// TwinCAT 3 PLC project UtilitiesLib
// Title: IBF_Utilities
// Company: Industrial Brains B.V.
// ProjectVersion: 2.0.0.0
// Description: Utilities library contains all basic utilities needed like system variables, messages, parameters etc.
// ProgramVersion: 3.1.4022.4
// libraries:
//   Tc2_Standard, * (Beckhoff Automation GmbH)
//   Tc2_System, * (Beckhoff Automation GmbH)
//   Tc2_Utilities, * (Beckhoff Automation GmbH)
//   Tc3_EventLogger, * (Beckhoff Automation GmbH)
//   Tc3_Module, * (Beckhoff Automation GmbH)
// project tree:
//   Avarage/ FB_RollingAverageLREAL.TcPOU, FB_RollingAverageTime.TcPOU, F_AverageLREAL.TcPOU, F_AverageTime.TcPOU
//   BaseFunctions/ FB_Base.TcPOU, FB_Base_WithEvent.TcPOU, FB_FunctionBase.TcPOU, FB_FunctionBase_WIthEvent.TcPOU
//   Compare/Functions/ Between.TcPOU, Between360deg.TcPOU
//   Conversion/ DegS_To_Rpm.TcPOU, DegS_To_Rpm_And_MMin.TcPOU, Grey_To_Bin.TcPOU, MMin_To_Rpm_And_DegS.TcPOU, Rpm_To_DegS.TcPOU
//   FaultsAndMessages/Functions/ FB_EventHandler.TcPOU, Fb_FaultHandler.TcPOU, FB_OperatorMessageDisplay.TcPOU
//   General/DataTypes/ Udt_TimerBandwith.TcDUT
//   GVLs/ DataManager.TcGVL, GVL_FixedValues.TcGVL, GVL_Message.TcGVL, GVL_Parameters.TcGVL, Sys_Variables.TcGVL
//   FaultsAndMessages/DataTypes/ E_ComponentTypes.TcTLEO, E_Locations.TcTLEO, E_MessageNumbers.TcTLEO, E_FaultTypes.TcTLEO, UDT_Fault.TcDUT
//   FaultsAndMessages/ Param_Messages.TcGVL
//   MovePathCalculations/ fAccDecCalc.TcPOU (not stored)
//   Parameter/DataTypes/Old/ UDT_Parameter_1.TcDUT, Udt_ParameterRetain.TcDUT, Udt_Parameter_2.TcDUT, Udt_ParLog_Old.TcDUT
//   Parameter/DataTypes/ Udt_ParameterId.TcDUT, Udt_Parameter.TcDUT
//   Parameter/Functions/ FB_ParameterHandler.TcPOU, Fb_ParLogging.TcPOU, F_ParToCsvLine.TcPOU
//   PathFunctions/ F_FBNameFromPath.TcPOU, F_GetLevelFromPath.TcPOU
//   Positions/FunctionBlocks/ FB_PositionTrigger_Old.TcPOU, FB_PositionTrigger.TcPOU
//   Positions/Functions/ F_AccDecDistanceFromTime.TcPOU, F_AccDecDistanceFromVelo.TcPOU, F_PosCheck.TcPOU, F_TopVelocityFromTime.TcPOU, F_TriggerPosOffset.TcPOU
//   StepFunctions/ FB_CycleTrigger.TcPOU (not stored), FB_Step.TcPOU
//   System/Functions/DataManagement/ FB_PersistentDataManager.TcPOU
//   System/Functions/ Fb_SystemVariables.TcPOU
//   / Utilities_CD.TcCD (not stored)

// ---- General/DataTypes/Udt_TimerBandwith.TcDUT
TYPE Udt_TimerBandwith :
STRUCT
	Minimal	:LREAL;// Timer values, Minimum time
	Nominal	:LREAL;// timer values, nominal time
	Maximum	:LREAL;// Timer values, Maximum time
END_STRUCT
END_TYPE

// ---- FaultsAndMessages/DataTypes/E_ComponentTypes.TcTLEO
{attribute 'qualified_only'}
{attribute 'strict'}
{attribute 'to_string'}
TYPE E_ComponentTypes :
(
	// No entry
		NA			:= 0,
	// Actuators 
		Cylinder 	:= 10,
		Axis		:= 11,
		Heaters		:= 12,
	// Buttons 
		EstopButton	:= 20,
		EstopBumper	:= 21,	
		Pushbutton 	:= 22,
		Switch		:= 23,
	// I/O
		SafeIO		:= 30,
		Rio_Box		:= 31,
		Rio_Slot	:= 32,
		Encoder		:= 33,
		DiInput		:= 34,
		AnInput		:= 35,
		DiOutput	:= 36,
		AnOutput	:= 37,
	// Drive
		ServoDrive 	:= 40,
	// Operation
		HMI			:= 50,
		RemoteOS	:= 51,
		RemoteDB	:= 52,
	// Assemblies
		Assembly 	:= 60,
		SubAssembly	:= 61,
	// functions
		MainProgram		:= 100,
		StepProgram		:= 101,
		FunctionBlock	:= 102 
)UDINT;
END_TYPE

// ---- FaultsAndMessages/DataTypes/E_Locations.TcTLEO
{attribute 'qualified_only'}
{attribute 'strict'}
TYPE E_Locations :
(
	MainPLC,
	MainPower_230V, 
	MainPower_24V, 
	MainAirSupply,
	MainScreen,
	MainIO,
	RemoteIO
);
END_TYPE

// ---- FaultsAndMessages/DataTypes/E_MessageNumbers.TcTLEO
{attribute 'qualified_only'}
{attribute 'strict'}
TYPE E_MessageNumbers :
(
	// no messages
		NA_NoMessage		:= 0, // no message active
	// System faults
		FF_Unknown 			:= 1, // unknown error occured 
		FF_NoCommunication 	:= 2, // no communication detected
		FF_ComunicationFault:= 3, // Communication error detected (does not match expected com)
		FF_Overload			:= 4, // hardware overload detected
		FF_EncoderFault		:= 5, // encoder signal incorrect or not present
		FF_SlaveFault		:= 6, // slave system is has active fatal fault
		FF_AxisFault		:= 7, // Axis fault feedback
		FF_DriveFault		:= 8, // Axis drive fault
		FF_Collision		:= 9, // Collision detected between 2 or more parts of the machine
	// Hardware faults
		CF_FeedbackFault		:= 100,	// Hardware feedback is does not match expected
		CF_WrongDirection		:= 101, // Hardware moving in incorrect direction
		CF_MoveToFast			:= 102, // Hardware movement completion time is lower then minimum
		CF_MoveToSlow			:= 103, // hardware movement maximum time was exceeded
		CF_WrongPosition		:= 104,	// Hardware is at different position then expected
		CF_Obstruction			:= 105, // Obstruction detected in movement path
	// Missing conditions
		MC_WaitingForproduct	:= 200,	// Waiting for product
		MC_WaitingForOperator	:= 201, // Waiting for operator action
		MC_WaitingForModule		:= 202,	// Waiting for other module
		MC_WaitingForMaster		:= 203, // Waiting Waiting for master
		MC_WaitingForSlave		:= 204, // waiting for slave
		MC_WrongPosition		:= 205, // Action or command not possible in current position
	// Operator messages
		OM_AlmostEmpty			:= 300, // product is almost empty refil is required
		OM_Finished 			:= 301, // product or action is finished
		OM_ready				:= 302, // ready for new task
	// Test Messages
		FF_MessageTest			:= 900, // Fatal fault message test
		CF_MessageTest			:= 901, // Cycle fault message test
		MC_MessageTest			:= 902, // Missing condition message test
		OM_MessageTest			:= 903	// Operator message test
)UDINT;
END_TYPE

// ---- FaultsAndMessages/DataTypes/E_FaultTypes.TcTLEO
{attribute 'qualified_only'}
{attribute 'strict'}
{attribute 'to_string'}
TYPE E_FaultTypes :
(
	NA	:= 0, // Not applicable
	OM 	:= 1, // Operator message
	MC	:= 2, // Missing condition
	CF	:= 3, // Cycle Fault
	FF	:= 4, // Fatal fault
	OW  := 5  // Operator warning
)UDINT;
END_TYPE

// ---- FaultsAndMessages/DataTypes/UDT_Fault.TcDUT
TYPE UDT_Fault :
STRUCT
	// active 
		Active 			: BOOL 				:= FALSE;
	// Message type
 		FaultType 		: E_FaultTypes 		:= E_FaultTypes.NA; // Type of message
	// Message Id number used for translation
		MessageNumber 	: UDINT				:= 0; // message number
		LocationNumber	: UDINT 			:= 0; // message number array ([1]= System, [2]= Module,[3]= sub module, [4]= Component)
	// Message discription
		Discription 	: STRING 			:= ''; // Message text discription in english (service personel only)
	// Location
		LocationName	: STRING			:= ''; // Location discription name
		ComponentType 	: E_ComponentTypes 	:= E_ComponentTypes.NA; // Part type discription
	// Time stamp
		StartTime		: DATE_AND_TIME 	:= DT#2020-1-1-00:00:00 ; // Time and date of message occurence
		EndTime			: DATE_AND_TIME		:= DT#2020-1-1-00:00:00 ; // Time and date of message end
	// Module number
		nModuleID		: UDINT 			; // module reference number used for fault, enable, reset, and safety functions (default := 1, 0 = main system)
	// CompleteFaultnumber for visualization
		FullFaultId		: STRING 			:= 'NA.0.0.0'; // Full fault id for use in HMI is writen by fault function [fault type, message#, location#,ComponentType]
END_STRUCT
END_TYPE

// ---- Parameter/DataTypes/Old/UDT_Parameter_1.TcDUT
TYPE UDT_Parameter_1 EXTENDS Udt_ParameterRetain:
STRUCT
	Name		: STRING	; // Parameter data, Parameter name
	Number		: INT		; // Parameter data, Parameter number
	Par_TYPE	: STRING	; // Parameter data, Type of parameter [Mpar, Cpar, Opar, Ppar]
	Discription	: STRING	; // Parameter data, Parmater discription
	Factory		: LREAL		; // Parameter data, Factory standard value
	Maximum		: LREAL		; // Parameter data, Maximum parameter value
	Minimum		: LREAL		; // Parameter data, Minimum parameter value
	Unit		: STRING	; // Parameter data, Unit of measurement
END_STRUCT
END_TYPE

// ---- Parameter/DataTypes/Old/Udt_ParameterRetain.TcDUT
TYPE Udt_ParameterRetain :
STRUCT
	PrepValue	: LREAL		; // Parameter data, prepared value
	Value		: LREAL		; // Parameter data, Current (active) parameter value
	Saved		: LREAL		; // Parameter data, Saved value or standard setpoint
	LastChange	: DT		; // Parameter data, Date of last change
END_STRUCT
END_TYPE

// ---- Parameter/DataTypes/Old/Udt_Parameter_2.TcDUT
TYPE Udt_Parameter_2 :
STRUCT
	bActive		: BOOL 	; // True if parameter is active in machine 
	IndexNumber	: UDINT	; // [Column 0] Array row index number  
	Number		: INT	; // [Column 1]Parameter data, parameter number
	Name		: STRING; // [Column 2]Parameter data, Parameter name
	Par_Type	: STRING; // [Column 3]Parameter data, Type of parameter [Mpar, Cpar, Opar, Ppar]
	Discription	: STRING; // [Column 4]Parameter data, Parmater discription
	Factory		: LREAL	; // [Column 5]Parameter data, Factory standard value
	Maximum		: LREAL	; // [Column 6]Parameter data, Maximum parameter value
	Minimum		: LREAL	; // [Column 7]Parameter data, Minimum parameter value
	Unit		: STRING; // [Column 8]Parameter data, Unit of measurement
	Value		: LREAL	; // [Column 9]Parameter data, Current (active) parameter value
	Saved		: LREAL	; // [Column 10]Parameter data, Saved value or standard setpoint
	bCmdTeach	: BOOL	; // Teach command for devices 
	bCmdSave	: BOOL 	; // Command to parameter handler to save the parameter
//	LastChange	: DT	; // [Column 11]Parameter data, Date of last change
END_STRUCT
END_TYPE

// ---- Parameter/DataTypes/Old/Udt_ParLog_Old.TcDUT
TYPE Udt_ParLog_Old :
STRUCT
	ParList		: ARRAY [1..GVL_Parameters.MAX_PARAMETERS] OF Udt_Parameter_2 ; // active parameter list
END_STRUCT
END_TYPE

// ---- Parameter/DataTypes/Udt_ParameterId.TcDUT
TYPE Udt_ParameterId :
STRUCT
	nNumber		: UDINT 	:= 0 	; // parameter number
	sName		: STRING 	:= 'NA' ; // parameter name
	sType		: STRING 	:= 'Ppar'	; // parameter type 
	pParameter	: POINTER TO Udt_Parameter ; // pointer to parameter
END_STRUCT
END_TYPE

// ---- Parameter/DataTypes/Udt_Parameter.TcDUT
TYPE Udt_Parameter :
STRUCT PERSISTENT
	nNumber		: UDINT	 	:= 0				; // [Column 0]Parameter data, parameter number
	sName		: STRING	:= 'No parameter' 	; // [Column 1]Parameter data, Parameter name
	sType		: STRING	:= 'PPar'			; // [Column 2]Parameter data, Type of parameter [Mpar, Cpar, Opar, Ppar]
	sDiscription: STRING	:= 'No parameter selcted'; // [Column 3]Parameter data, Parmater discription
	fFactory	: LREAL		:= 0				; // [Column 4]Parameter data, Factory standard value
	fMaximum	: LREAL		:= 0				; // [Column 5]Parameter data, Maximum parameter value
	fMinimum	: LREAL		:= 0				; // [Column 6]Parameter data, Minimum parameter value
	sUnit		: STRING	:= 'na'				; // [Column 7]Parameter data, Unit of measurement
	fValue		: LREAL		:= 0				; // [Column 8]Parameter data, Current (active) parameter value
	fSaved		: LREAL		:= 0				; // Parameter data, Saved value or standard setpoint
	fPrepared	: LREAL 	:= 0				; // Parameter data, Prepared value from teach function 
	bCmdTeach	: BOOL		:= FALSE			; // Teach command for devices 
	bAccepted	: BOOL 		:= FALSE 			; // Paramer value has been accepted
END_STRUCT
END_TYPE

// ---- GVLs/DataManager.TcGVL
{attribute 'qualified_only'}
VAR_GLOBAL
	FbPersistentManager : FB_PersistentDataManager ;
END_VAR

// ---- GVLs/GVL_FixedValues.TcGVL
{attribute 'qualified_only'}
VAR_GLOBAL
	nINTMAXVALUE	: INT := 32767 		; // Integer maximum value 32767
	nINTMINVALUE	: INT := -32767		; // intiger minimum value -32767
	nDINTMAXVALUE	: DINT:= 2147483647 ; // Double integer maximum value 2,147,483,647
	nDINTMINVALUE	: DINT:= -2147483647; // Double integer minimum value -2,147,483,647
END_VAR

// ---- GVLs/GVL_Message.TcGVL
{attribute 'qualified_only'}
VAR_GLOBAL
	bResetFaults		: BOOL 	:= FALSE	; // Reset system faults 
	bCmdSnoozeMessage	: BOOL 	:= FALSE	; // Snooze message display
	bHideFaults			: BOOL 	:= FALSE 	; // Display fault message popup on screen (when MC, CF of FF are active)
	bHideReset			: BOOL 	:= FALSE 	; // Hide reset button in display unless CF of FF is active 
	bHideWarnAck		: BOOL	:= FALSE	; // Hide the warning acknowledge button on the HMI (when OW is active)
	bAckWarnings		: BOOL	:= FALSE	; // Acknowledge the warning(s)
	arActiveFaults 		: ARRAY [0..Param_Messages.nMAX_MESSAGES_SHOWN] OF UDT_Fault ; // Active faults overview for showing in HMI
	sOPeratorMessage	: STRING ;	// operator message for displaying non vital machine data
END_VAR
VAR_GLOBAL CONSTANT 
	tMESSAGESNOOZEDURATION	: TIME 	:= T#5s ; // duration of message snooze after button press 
END_VAR

// ---- GVLs/GVL_Parameters.TcGVL
{attribute 'qualified_only'}
VAR_GLOBAL
	fbParameterHandler		: Fb_ParLogging ; // Default parameter handler for visualisation and file handling
	sPARLIST_FILE			: T_MaxString 		:= 'D:\Parameters\ParameterList.csv';(* CSV destination file path and name *)
	sPARLOG_FILE			: T_MaxString 		:= 'D:\Parameters\ParameterLog.csv';(* CSV destination file path and name *)
END_VAR
VAR_GLOBAL CONSTANT
	MAX_PARAMETERS 			: UDINT := 1000	;
	PAR_COLUMNS 			: UDINT := 8	;
	MAX_CSV_FIELD_LENGTH	: UDINT := 100	;
	sNetId					: T_AmsNetID		:= '' ;
END_VAR

// ---- GVLs/Sys_Variables.TcGVL
(* System variables *)
{attribute 'qualified_only'}
VAR_GLOBAL
// SystemFuntion
	fbSystemVariables : Fb_SystemVariables ;
	AlwaysOn		:BOOL 			;// System variable, Always on bit
	AlwaysOff		:BOOL 			;// System variable, Always off bit
	BlinkFast		:BOOL 			;// System variable, Blink fast bit 1sec 
	BlinkSlow		:BOOL 			;// System variable, Blink slow bit 2 sec
	Pulse1Sec		:BOOL 			;// System variable, Pulse 1 cycle every second
	Pulse100ms		:BOOL 			;// System variable, pulse 1 cycle every 100 ms
	SystemTime		:DT				; // System variable, Windows system time
	TimeZoneId		:E_TimeZoneID 	; // System variable, time zone Id 
	HeartBeat		:BOOL 			;// System Variable, Main system heartbeat 0.5 sec on 0.5 sec off
END_VAR

// ---- FaultsAndMessages/Param_Messages.TcGVL
{attribute 'qualified_only'}
VAR_GLOBAL CONSTANT
	nMAX_MESSAGES_SHOWN 	: UDINT := 10 	;
	nMAX_MESSAGE_HISTORY	: UDINT := 1000 ;
	nMAX_CSV_FIELD_LENGTH	: UDINT := 100	;
	tMESSAGE_TIMEOUT		: TIME 	:= T#5S ;
	sLOGFILE_PATH			: STRING:= '\Hard Disk\TwinCAT\3.1\Boot\FaultLogs\'	;
	sLOGFILE_NAME			: STRING:= 'Faultlog' 		; // Message log destination file
	nMESSAGE_COLUMNS		: UDINT := 8 ;
END_VAR

// ---- System/Functions/DataManagement/FB_PersistentDataManager.TcPOU
FUNCTION_BLOCK FB_PersistentDataManager
VAR_INPUT
END_VAR
VAR_OUTPUT
END_VAR
VAR
	FbWritePersistentData : FB_WritePersistentData ;
	cmdWrite : BOOL := FALSE ;
	TOfWriteInterval	: TOf ;
	CmdWriteFromTime	: BOOL ; 
	TestjeWritten		: BOOL ;
END_VAR

// ===== persistent write interval =====
 TOfWriteInterval(	IN := cmdWrite OR NOT TOfWriteInterval.Q,
	 				PT	:= T#5M  );

IF NOT TOfWriteInterval.Q THEN 
	cmdWrite := TRUE ;
END_IF

// ===== write persistent data =====
	FbWritePersistentData ( PORT 	:= 851,
							START 	:= CmdWrite,
							TMOUT 	:= T#1S,	
							mode 	:= E_PersistentMode.SPDM_VAR_BOOST );	

IF cmdWrite AND FbWritePersistentData.BUSY THEN 
	cmdWrite := FALSE ;
END_IF

METHOD PUBLIC Write : BOOL
VAR_INPUT
END_VAR
IF NOT FbWritePersistentData.BUSY THEN 
	cmdWrite := TRUE ;
ELSE 
	Write := TRUE ;
END_IF
END_METHOD

END_FUNCTION_BLOCK

// ---- Parameter/Functions/Fb_ParLogging.TcPOU
FUNCTION_BLOCK PUBLIC Fb_ParLogging EXTENDS FB_ParameterHandler
VAR_OUTPUT
	stParLog		: Udt_ParLog_Old ; // active parameter list
	bReadBusy		: BOOL		:= FALSE	; // File acces Bussy
	bWriteBusy		: BOOL 		:= FALSE	; // file write bussy
	bError			: BOOL		:= FALSE	; // File acces error
	nErrId			: UDINT		:= 0		; // File acces error Id
	nRow	 		: UDINT 	:= 0		;(* Row number (record) *)
	nColumn			: UDINT 	:= 0		;(* Column number (record field) *)
	nInitStep		: UDINT 	:= 0 		; // Initialization step
END_VAR
VAR
	// ====== Compare array =====
		arFileParameters		: ARRAY [1..GVL_Parameters.MAX_PARAMETERS] OF Udt_Parameter;
		nNumberOfParFromFile	: UDINT; // Number of parameters read from file
		nNumberOfChanges		: UDINT; // Number of parameter changes 
		arChangeLog				: ARRAY [0..(GVL_Parameters.MAX_PARAMETERS * 2)] OF STRING ; // Parameter change log 
	// ====== Internal commands ======
		bCmdParFileWrite	: BOOL ; // write alle parameters to .csv file
		bCmdParLogWrite		: BOOL ; // write all changes to .csv file
		bCmdParFileRead		: BOOL ; // Read all parameters from .csv file 
		StParameter			: UDT_Parameter_1 ;
	// ====== File headers ======
		sCsvFileHeader : STRING := 'NUMBER;NAME;TYPE;DISCRIPTION;FACTORY;MAXIMUM;MINIMUM;UNIT;VALUE$L';
	// ====== internal status ======
		bInitOK				: BOOL 	:= FALSE ; // init has been done succesfully
		bFileNotFound		: BOOL 	:= FALSE ; // Parameter file has not been found 
		bParCountDiference	: BOOL 	:= FALSE ; // The number of parameters from file does not match machine 
		bParNumberDiference	: BOOL 	:= FALSE ; // The parameters from file do not match machine
		nDiferenceRow		: UDINT	:= 0	 ; // The file array row number in which diferences were found
 
	// ====== Current step =====
		nReadStep			: INT 	:= 0 	; // File read stepper
		nLogStep			: INT 	:= 0 	; // File logging step
		nWriteStep			: INT 	:= 0 	; // File Write stepper

	// ====== Read variables ======
		hFile				: UINT	:= 0;(* File handle of the source file *)
		cbField				: UDINT	;(* Number of bytes in field buffer *)

	// ====== Read variables ======
		sCSVLine			: T_MaxString := '';(* Single CSV text line (row, record), we are using string as record buffer (your are able to see created fields) *)
		sCSVField			: T_MaxString := '';(* Single CSV field value (column, record field) *)
		sCSVFieldString		: T_MaxString := '';// CSV field converted into string
	// ====== Functions ======
		fbFileOpenForRead	: FB_FileOpen	;(* Opens file *)
		fbFileOpenForWrite	: FB_FileOpen	;(* Opens file *)
		fbFileOpenForLog	: FB_FileOpen	;(* Opens file *)
		fbFileClose			: FB_FileClose	;(* Closes file *)
		fbFileGets			: FB_FileGets	;(* Reads one record (line) *)
		fbFilePuts			: FB_FilePuts	;(* Writes one record (line) *)
		fbReader			: FB_CSVMemBufferReader;(* Helper function block used to parse CSV data bytes (single record line) *)
		fbWriter			: FB_CSVMemBufferWriter;(* Helper function block used to create CSV data bytes (single record line) *)
	
	// Par Read timeout 
		TonParWriteTimeout	: TON := (PT := T#5S) ; // Timeout for parameter read
		TonParreadTimeout	: TON := (PT := T#5S) ; // Timeout for parameter read
		
END_VAR

SUPER^();

// ===== init =====
	IF NOT binitok THEN 
		RETURN;
	ELSE 
		CmdParWriteToFile();
		CmdParLoadFromFile();
	END_IF

METHOD PRIVATE CmdParLoadFromFile : BOOL
VAR_INPUT
END_VAR
VAR 
	i : UDINT ;
	fTempValue	: LREAL ; // Tomporary value to be placed in save value
END_VAR
IF ExecFileRead() THEN 
	;
ELSE
	RETURN;
END_IF

// Compare Parameter counters 
IF nNumberOfParameters <> nNumberOfParFromFile THEN
	bParCountDiference := TRUE ;
ELSE 
	bParCountDiference := FALSE ;
END_IF

// Compare Parameter from file with parameters in machine then write from file to machine
bParNumberDiference := FALSE ;
nDiferenceRow		:= 0 ;
IF NOT bParCountDiference THEN 
	FOR i := 1 TO nNumberOfParameters DO
		IF arParameters[i].nNumber <> arFileParameters[i].nNumber THEN
			bParNumberDiference := TRUE ;
			nDiferenceRow		:= i ;
			CONTINUE;
		ELSE
			IF (arParameters[i].pParameter^.fValue <> arFileParameters[i].fValue) THEN 
				fTempValue := arParameters[i].pParameter^.fValue;  
			ELSE
				fTempValue := 0;
			END_IF
			arParameters[i].pParameter^			:= arFileParameters[i];
			arParameters[i].pParameter^.fSaved 	:= fTempValue;
		END_IF
	END_FOR
END_IF 

CmdParLoadFromFile := TRUE ;
END_METHOD

METHOD PRIVATE CmdParWriteToFile : BOOL
VAR_INPUT
END_VAR
VAR
	i : UDINT ;
	sDTString : STRING ;
END_VAR

IF bCmdParFileWrite THEN 
	FOR i := 1 TO nNumberOfParameters DO
(*			IF 	NOT bFileNotFound AND
				(arFileParameters[i].fValue <> arParameters[i].pParameter^.fValue OR
				arFileParameters[i].fFactory <> arParameters[i].pParameter^.fFactory) THEN
					sDTString := DT_TO_STRING(Sys_Variables.SystemTime);
					sDTString := STRING_TO_CSVFIELD(sdtstring,TRUE);
					arChangeLog[nNumberOfChanges*2] := CONCAT(sDTString,F_ParToCsvLine( arFileParameters[i],));
					arChangeLog[(nNumberOfChanges*2)+1] := CONCAT( ';', STR2 := F_ParToCsvLine( arParameters[i].pParameter^)); 
					bCmdParLogWrite 	:= TRUE ;
					nNumberOfChanges	:= LIMIT(0,nNumberOfChanges + 1, nNumberOfParameters); 
			END_IF 
*)
			// Save current actual value for later restore
			IF arParameters[i].pParameter^.fValue <> arFileParameters[i].fValue THEN
				arParameters[i].pParameter^.fSaved := arFileParameters[i].fValue ;
			END_IF
			arFileParameters[i] := arParameters[i].pParameter^ ;
	END_FOR
END_IF

//IF nNumberOfChanges > 0 AND NOT bParCountDiference THEN 
//	ExecWriteToLog();
//END_IF
CmdParWriteToFile := ExecFileWrite();
END_METHOD

METHOD PUBLIC CmdSavePar : BOOL
VAR_INPUT
END_VAR
bCmdParFileWrite := TRUE ;

CmdSavePar := bWriteBusy ;
END_METHOD

METHOD PRIVATE ExecFileRead : BOOL
VAR_INPUT
END_VAR
VAR
	i : UDINT := 0 ;
END_VAR
// ===== Wait for command =====
	IF bCmdParFileRead OR bReadBusy THEN 
		;
	ELSE
		RETURN ;
	END_IF

// ===== prepare for file read =====
	CASE nReadStep OF
		0:	(* Wait for rising edge at bRead variable *)
			bReadBusy		:= TRUE;
			bFileNotFound	:= FALSE ;
			bCmdParFileRead := FALSE ;
			bError			:= FALSE;
			nErrId			:= 0;
			hFile			:= 0;
			nRow			:= 0;
			nColumn			:= 0;
			nReadStep 			:= 1;
	
		1:	(* Open source file *)
			fbFileOpenForRead(  bExecute := FALSE  );
			fbFileOpenForRead( sNetId := GVL_Parameters.sNetId, sPathName := GVL_Parameters.sPARLIST_FILE, nMode := FOPEN_MODEREAD OR FOPEN_MODETEXT,(* Open file in text mode! *)
						ePath := PATH_GENERIC, bExecute := TRUE );
			nReadStep := 2;
	
		2:(* Wait until open not busy *)
			fbFileOpenForRead( bExecute := FALSE, bError => bError, nErrID => nErrID, hFile => hFile );
			IF NOT fbFileOpenForRead.bBusy THEN
				IF NOT fbFileOpenForRead.bError THEN
					nReadStep := 3;
				ELSE(* Error: file not found? *)
					bFileNotFound := TRUE ;
					nReadStep := 100;
				END_IF
			END_IF
		3:	(* Read single line (record) *)
			fbFileGets( bExecute := FALSE );
			fbFileGets( sNetId := GVL_Parameters.sNetId, hFile := hFile, bExecute := TRUE );
			nReadStep := 4;
		4:(* Wait until read not busy *)
			fbFileGets( bExecute := FALSE, bError => bError, nErrID => nErrID, sLine => sCSVLine );
			IF NOT fbFileGets.bBusy THEN
				IF NOT fbFileGets.bError THEN
					IF fbFileGets.bEOF THEN
						nReadStep 				:= 10;(* End of file reached => Close source file *)
					ELSE
						(* FB_FileGets returns text line without the CR (carriage return) character.
						We have to restore the CR character (replace the $L character with $R$L characters) *)
						IF RIGHT( sCSVLine, 1 ) = '$L' THEN
							sCSVLine := REPLACE( sCSVLine, '$R$L', 2, LEN( sCSVLine ) );
						END_IF
						nReadStep := 5;
					END_IF
				ELSE(* Error *)
					nReadStep := 100;
				END_IF
			END_IF
		5:(* Parse single line (record) *)
			fbReader.eCmd := eEnumCmd_First;(* Read first field value *)
			REPEAT
				fbReader( pBuffer := ADR( sCSVLine ), cbBuffer := SIZEOF( sCSVLine ), getValue => sCSVField );
				IF fbReader.bOk THEN
					fbReader.eCmd := eEnumCmd_Next;(* Read next field value *)
					IF ( nRow <= GVL_Parameters.MAX_PARAMETERS ) AND nRow > 0 THEN
						IF ( nColumn <= GVL_Parameters.PAR_COLUMNS ) THEN
							sCSVFieldString	:= CSVFIELD_TO_STRING( sCSVField, TRUE);
							CASE nColumn OF
									0: // Parameter number [Udint]	
										arFileParameters[nRow].nNumber		:= STRING_TO_UDINT(sCSVFieldString); 						
									1: // Parameter Name [string]
										arFileParameters[nRow].sName 		:= sCSVFieldString;							
									2: // Parameter type [String]
										arFileParameters[nRow].sType 		:= sCSVFieldString;	
									3: // Parameter discription [string]
										arFileParameters[nRow].sDiscription:= sCSVFieldString;						
									4: // Parameter factory value [LREAL]
										arFileParameters[nRow].fFactory	:= STRING_TO_LREAL(sCSVFieldString);							
									5: // Parameter maximum value [LREAL]
										arFileParameters[nRow].fMaximum	:= STRING_TO_LREAL(sCSVFieldString);							
									6: // Parameter minimum value[LREAL]
										arFileParameters[nRow].fMinimum	:= STRING_TO_LREAL(sCSVFieldString);							
									7: // Parameter unit {String]
										arFileParameters[nRow].sUnit 		:= sCSVFieldString;							
									8: // Parameter value [LREAL]
										arFileParameters[nRow].fValue		:= STRING_TO_LREAL(sCSVFieldString);							
							ELSE
								;
							END_CASE
						END_IF
					END_IF
					nColumn := nColumn + 1;(* Increment number of read columns *)
					IF fbReader.bCRLF THEN(* CRLF == TRUE => End of reacord reached *)
						nNumberOfParFromFile := nRow;
						nRow 		:= nRow + 1;(* Increment number of read records *)
						nColumn 	:= 0;(* Reset number of columns *)
					END_IF
				ELSE(* Error: End of record reached or all fields read *)
					nReadStep := 3;(* Try to read next line *)
				END_IF
			UNTIL NOT fbReader.bOk
			END_REPEAT
		10:	(* Close source file *)
			fbFileClose( bExecute := FALSE );
			fbFileClose( sNetId := GVL_Parameters.sNetId, hFile := hFile, bExecute := TRUE );
			nReadStep := 11;
	
		11:(* Wait until close not busy *)
			fbFileClose( bExecute := FALSE, bError => bError, nErrID => nErrID );
			IF ( NOT fbFileClose.bBusy ) THEN
				hFile := 0;
				nReadStep := 100;
			END_IF
		100: (* Error or ready nReadStep => cleanup *)
			IF ( hFile <> 0 ) THEN
				nReadStep := 10; (* Close the source file *)
			ELSE
				bReadBusy := FALSE;
				ExecFileRead := TRUE ;
				nReadStep := 0;	(* Ready *)
			END_IF
	END_CASE
	
	TonParreadTimeout(IN := bReadBusy);
	bError S= TonParreadTimeout.Q;
END_METHOD

METHOD INTERNAL ExecFileWrite : BOOL
VAR_INPUT
END_VAR
// ===== Wait for command =====
	IF bCmdParFileWrite OR bWriteBusy THEN 
		;
	ELSE
		RETURN ;
	END_IF

// ===== Start file write =====
	CASE nWriteStep OF
		0:	(* Wait for rising edge at bWrite variable *)
				bFileNotFound		:= FALSE ;
				bParCountDiference	:= FALSE ;
				bWriteBusy 			:= TRUE;
				bCmdParFileWrite	:= FALSE ;
				bError				:= FALSE;
				nErrId				:= 0;
				hFile				:= 0;
				nRow				:= 0;
				nWriteStep 				:= 1;
		1:	(* Open source file *)
			fbFileOpenForWrite(  bExecute := FALSE  );
			fbFileOpenForWrite( sNetId := GVL_Parameters.sNetId, sPathName := GVL_Parameters.sPARLIST_FILE, nMode := FOPEN_MODEWRITE OR FOPEN_MODETEXT,(* Open file in TEXT mode! *)
						ePath := PATH_GENERIC, bExecute := TRUE );
			nWriteStep := 2;
		2:(* Wait until open not busy *)
			fbFileOpenForWrite( bExecute := FALSE, bError => bError, nErrID => nErrID, hFile => hFile );
			IF NOT fbFileOpenForWrite.bBusy THEN
				IF NOT fbFileOpenForWrite.bError THEN
					nWriteStep := 3;
				ELSE(* Error: file not found? *)
					nWriteStep := 100;
				END_IF
			END_IF
	
		3:(* Convert one PLC parameter field to CSV format *)
			// Go column by column to avoid return strings that are too long
			// TODO test (default string constructor is 80 characters, but can be extended to <?>)
			IF nRow = 0 THEN 
				sCSVLine := sCsvFileHeader;
			ELSE
				sCSVLine := F_ParToCsvLine(stParameter := arFileParameters[nRow], nColumn := nColumn);
			END_IF
			nWriteStep := 4 ;
		4:	(* Write single Field *)
			fbFilePuts( bExecute := FALSE );
			fbFilePuts( sNetId := GVL_Parameters.sNetId, hFile := hFile, sLine := sCSVLine, bExecute := TRUE );
			nWriteStep := 5;
		5:(* Wait until write not busy *)
			fbFilePuts( bExecute := FALSE, bError => bError, nErrID => nErrID );
			IF NOT fbFilePuts.bBusy THEN
				IF NOT fbFilePuts.bError THEN
					nWriteStep := 3;(* Write next record *)
					IF nRow = 0 OR nColumn = 8 THEN
						nColumn := 0 ;
						nRow := nRow + 1;
						IF nRow = nNumberOfParameters + 1 THEN
							nWriteStep := 10;
						END_IF;
					ELSE
						nColumn := nColumn + 1;
					END_IF
				ELSE(* Error *)
					nWriteStep := 100;
				END_IF
			END_IF
		10:	(* Close source file *)
			fbFileClose( bExecute := FALSE );
			fbFileClose( sNetId := GVL_Parameters.sNetId, hFile := hFile, bExecute := TRUE );
			nWriteStep := 11;
	
		11:(* Wait until close not busy *)
			fbFileClose( bExecute := FALSE, bError => bError, nErrID => nErrID );
			IF ( NOT fbFileClose.bBusy ) THEN
				hFile := 0;
				nWriteStep := 100;
			END_IF
	
		100: (* Error or ready nWriteStep => cleanup *)
			IF ( hFile <> 0 ) THEN
				nWriteStep := 10; (* Close the source file *)
			ELSE
				bParCountDiference 	:= FALSE ;
				bWriteBusy 			:= FALSE;
				ExecFileWrite		:= TRUE ;
				nWriteStep 			:= 0;	(* Ready *)
			END_IF
	
	END_CASE
	
	TonParWriteTimeout(IN := bWriteBusy);
	bError	S= TonParWriteTimeout.Q ;
	

ExecFileWrite := TRUE ;
END_METHOD

METHOD PRIVATE ExecWriteToLog : BOOL
VAR_INPUT
END_VAR
VAR
	sTempField : STRING ;
END_VAR
// ===== Wait for command =====
	IF bWriteBusy OR bCmdParLogWrite THEN 
		;
	ELSE
		RETURN ;
	END_IF

// ===== Start file write =====
CASE nLogStep OF
	0:	(* Wait for rising edge at bWrite variable *)
			bWriteBusy 			:= TRUE;
			bCmdParLogWrite	:= FALSE ;
			bError				:= FALSE;
			nErrId				:= 0;
			hFile				:= 0;
			nRow				:= nNumberOfChanges * 2; // Twice the number of changes because old and new values are stored sequentially in teh same array
			nLogStep 			:= 1;
	1:	(* Open source file *)
		fbFileOpenForLog(  bExecute := FALSE  );
		fbFileOpenForLog( sNetId := GVL_Parameters.sNetId, sPathName := GVL_Parameters.sPARLIST_FILE, nMode := FOPEN_MODETEXT,(* Open file in TEXT mode! *)
					ePath := PATH_GENERIC, bExecute := TRUE );
		nLogStep := 2;
	2:(* Wait until open not busy *)
		fbFileOpenForLog( bExecute := FALSE, bError => bError, nErrID => nErrID, hFile => hFile );
		IF NOT fbFileOpenForLog.bBusy THEN
			IF NOT fbFileOpenForLog.bError THEN
				nLogStep := 3;
			ELSE(* Error: file not found? *)
				nLogStep := 100;
			END_IF
		END_IF

	3:(* Convert one PLC record to CSV format *)
		sCSVLine := arChangeLog[nRow];
		nLogStep := 4 ;
	4:	(* Write single text line *)
		fbFilePuts( bExecute := FALSE );
		fbFilePuts( sNetId := GVL_Parameters.sNetId, hFile := hFile, sLine := sCSVLine, bExecute := TRUE );
		nLogStep := 5;

	5:(* Wait until write not busy *)
		fbFilePuts( bExecute := FALSE, bError => bError, nErrID => nErrID );
		IF NOT fbFilePuts.bBusy THEN
			IF nRow = 0 THEN
				nNumberOfChanges := 0;
				nLogStep := 10;
			ELSIF NOT fbFilePuts.bError THEN
				arChangeLog[nRow] := ''; // Delete change from log
				nRow := nRow - 1;
				nLogStep := 3;(* Write next record *)
			ELSE(* Error *)
				nLogStep := 100;
			END_IF
		END_IF
	10:	(* Close source file *)
		fbFileClose( bExecute := FALSE );
		fbFileClose( sNetId := GVL_Parameters.sNetId, hFile := hFile, bExecute := TRUE );
		nLogStep := 11;

	11:(* Wait until close not busy *)
		fbFileClose( bExecute := FALSE, bError => bError, nErrID => nErrID );
		IF ( NOT fbFileClose.bBusy ) THEN
			hFile := 0;
			nLogStep := 100;
		END_IF

	100: (* Error or ready nLogStep => cleanup *)
		IF ( hFile <> 0 ) THEN
			nLogStep := 10; (* Close the source file *)
		ELSE
			bWriteBusy := FALSE;
			nLogStep := 0;	(* Ready *)
		END_IF
END_CASE
END_METHOD

METHOD PUBLIC Init : BOOL
VAR_INPUT
END_VAR
// Read parameters from .CSV file and check if load is valid

CASE nInitStep OF 
	0: //check if init has been done 
		bInitOK 	:= FALSE;
		nInitStep 	:= 10 ;
	10: // start File read
		bCmdParFileRead := TRUE ;
		nInitStep := 11; 
	11: // Execute file read 
		IF CmdParLoadFromFile() THEN 
			nInitStep := 12 ;
		END_IF
	12: // Check if read is valid 
		IF bFileNotFound OR bParCountDiference THEN 
			nInitStep := 20 ;
		ELSE 
			nInitStep := 100 ;
		END_IF
	20: // start File write
		bCmdParFileWrite:= TRUE ;
		nInitStep		:= 21 ;
	21: // Wait for file write to finish
		IF CmdParWriteToFile() THEN 
			nInitStep := 100 ;
		ELSIF bError THEN 
			nInitStep := 900 ; 
		END_IF 
	100: // Init ok 
		bInitOK 	:= TRUE ;
		Init		:= TRUE ;
		nInitStep	:= 0 ;
	900: // file fault	
		bInitOK := FALSE ;
		RETURN ;
	ELSE 
		;
END_CASE
END_METHOD

END_FUNCTION_BLOCK

// ---- Parameter/Functions/FB_ParameterHandler.TcPOU
FUNCTION_BLOCK PUBLIC FB_ParameterHandler
VAR_OUTPUT
	arParameters		: ARRAY [1..GVL_Parameters.MAX_PARAMETERS] OF Udt_ParameterId := [stDummyParId]; 
END_VAR
VAR
	nLookupIndex		: UDINT := 1;
	nNumberOfParameters : UDINT := 1;
	// parameter change commands
	bCmdLoadfactory		: BOOL 	:= FALSE; // Load factory value into prepared value 
	bCmdLoadFromPrevious: BOOL 	:= FALSE; // Load from saved previous value into prepared value
	bCmdTeach			: BOOL 	:= FALSE; // Start teaching function for selected parameter
	bCmdAcceptTeach		: BOOL 	:= FALSE ; // Accept the teach value
	// Dummy parameter when no parameters are added yet
	stDummyParId		: Udt_ParameterId ;
	// Memory 
	fValueOld			: LREAL	:= 0 ; // previous value
END_VAR

// call parameter change function 
ExecChangeParValues();

METHOD PUBLIC CmdAddParameter : BOOL
VAR_IN_OUT
	refParameter : Udt_Parameter ; // Parameter to add
END_VAR
VAR
	i 			: UDINT ;
	j			: UDINT ;
	stTempPar	: Udt_ParameterId ;
	bParFound	: BOOL 	:= FALSE ;
END_VAR
// Get number of parameters
FOR i := 1 TO GVL_Parameters.MAX_PARAMETERS DO
	IF arParameters[i].pParameter = 0 THEN
		nNumberOfParameters := i - 1;
		EXIT ;
	END_IF
END_FOR

// check if parameter is already added
FOR i := 1 TO nNumberOfParameters DO
	IF arParameters[i].nNumber = refParameter.nNumber THEN
		CmdAddParameter := TRUE;
 		RETURN ;
	END_IF
END_FOR
	
// Add parameter to array
nNumberOfParameters := nNumberOfParameters + 1; 
IF nNumberOfParameters <= GVL_Parameters.MAX_PARAMETERS THEN
	arParameters[nNumberOfParameters].nNumber		:= refParameter.nNumber 	;
	arParameters[nNumberOfParameters].sName			:= refParameter.sName	;
	arParameters[nNumberOfParameters].sType			:= refParameter.sType	;
	arParameters[nNumberOfParameters].pParameter 	:= ADR(refParameter)	;
	
	// (re)sort parameter list
	FOR i := 2 TO nNumberOfParameters BY 1 DO
		FOR j := 1 TO nNumberOfParameters -1 BY 1 DO
			IF (arParameters[j].nNumber > arParameters[j+1].nNumber)THEN
				stTempPar 			:= arParameters[j+1];
				arParameters[j+1]	:= arParameters[j];
				arParameters[j]		:= stTempPar ;
			END_IF
		END_FOR
	END_FOR	
	
	// set feedback
	CmdAddParameter S= arParameters[nNumberOfParameters].pParameter > 0 ;
ELSE
	CmdAddParameter := FALSE;	
END_IF
END_METHOD

METHOD ExecChangeParValues : BOOL
VAR
END_VAR
IF arParameters[nLookupIndex].pParameter <> 0 THEN 
	;
ELSE
	RETURN; 
END_IF

// Load values from default or saved
IF bCmdLoadfactory THEN 
	arParameters[nLookupIndex].pParameter^.fValue := arParameters[nLookupIndex].pParameter^.fFactory ;
	bCmdLoadfactory := FALSE ;
ELSIF bCmdLoadFromPrevious THEN
	arParameters[nLookupIndex].pParameter^.fValue := arParameters[nLookupIndex].pParameter^.fSaved ;
	bCmdLoadFromPrevious := FALSE ;
ELSIF bCmdAcceptTeach THEN 
	arParameters[nLookupIndex].pParameter^.fValue := arParameters[nLookupIndex].pParameter^.fPrepared ;
	bCmdAcceptTeach := FALSE ;
END_IF
END_METHOD

END_FUNCTION_BLOCK

// ---- Parameter/Functions/F_ParToCsvLine.TcPOU
FUNCTION F_ParToCsvLine : STRING // convert parameter into csv string (default UDt_Parameter setup)
VAR_INPUT
	stParameter : Udt_Parameter ; 
	nColumn		: UDINT ;
END_VAR
VAR
	sTempString : STRING ;
	sTempCsvField : STRING ;
END_VAR

CASE nColumn OF 
	0: // number
		sTempString := UDINT_TO_STRING(stParameter.nNumber);
	1: // name
		sTempString := stParameter.sName;
	2: // Type
		sTempString := stParameter.sType;
	3: // discription
		sTempString := stParameter.sDiscription;
	4: // factory
		sTempString := LREAL_TO_STRING(stParameter.fFactory);
	5: // maximum
		sTempString := LREAL_TO_STRING(stParameter.fMaximum);
	6: // minimum
		sTempString := LREAL_TO_STRING(stParameter.fMinimum);
	7: // Unit 
		sTempString := stParameter.sUnit;
	8: // value
		sTempString := LREAL_TO_STRING(stParameter.fValue);
	ELSE
		;
END_CASE
	sTempCsvField := STRING_TO_CSVFIELD(sTempString, FALSE);
IF nColumn < 8 THEN 
	sTempCsvField := CONCAT(StempCsvField,';');
ELSE
	sTempCsvField := CONCAT(StempCsvField,'$L');
END_IF

F_ParToCsvLine := sTempCsvField;

END_FUNCTION

// ---- System/Functions/Fb_SystemVariables.TcPOU
FUNCTION_BLOCK Fb_SystemVariables
VAR
	// **** Function blocks *****
		Fb_SystemTime: FB_LocalSystemTime ;
		Fb_TimerHbOn : Ton ; // Timer Heartbeat on
		Fb_TimerFast : Ton ; // Timer for fast blink bit
		Fb_TimerSlow : Ton ; // Timer for slow blink bit
		Fb_RisingPulse : R_Trig ; // Rinsing edge trigger function	
	// ***** internal Variables *****
		TimeStruct	: TIMESTRUCT ; // Time structure from system time function
		HeartbeatOn	: BOOL ; // heartbeat is on
		FlashFastOn	: BOOL ; // Fast Flash bit on
		FlashSlowOn	: BOOL ; // Flash slow bit on
	
		Fb_Timer100mSec : TON := (PT := T#100MS); // Timer for 100 ms pulse		
END_VAR

// ===== Get system time =====
	// ***** get windows system time *****
		Fb_SystemTime(	sNetID := '', 
						bEnable := TRUE, 
						dwCycle := 1,
						dwOpt := 0, 
						tTimeout := DEFAULT_ADS_TIMEOUT, 	
						systemTime => TimeStruct,
						tzID	=> Sys_Variables.TimeZoneId
						);
	// ****** convert to time of day format *****
		Sys_Variables.SystemTime := SYSTEMTIME_TO_DT(TIMESTR := TimeStruct) ;

// ===== Heartbeat generator =====
	Fb_TimerHbOn(In := NOT HeartbeatOn , PT:= T#1S, Q => HeartbeatOn);
	IF Fb_TimerHbOn.ET >= T#500MS THEN
		Sys_Variables.HeartBeat := TRUE ;
	ELSE
		Sys_Variables.HeartBeat := FALSE ;
	END_IF

// ===== one second pulse generator =====
	Fb_RisingPulse(Clk := HeartbeatOn, Q => Sys_Variables.Pulse1Sec);
	
// ===== 100ms pulse generation ======
	Fb_Timer100mSec( IN := NOT Sys_Variables.Pulse100ms, Q => Sys_Variables.Pulse100ms);

// ===== Flash fast bit =====
	Fb_TimerFast(In := NOT FlashFastOn, Pt := T#1S, Q => FlashFastOn);
	IF Fb_TimerFast.ET >= T#600MS THEN
		Sys_Variables.BlinkFast := TRUE;  
	ELSE
		Sys_Variables.BlinkFast := FALSE;  		
	END_IF
// ===== Flash Slow bit =====
	Fb_TimerSlow(In := NOT FlashSLowOn, Pt := T#2S, Q => FlashSlowOn);
	IF Fb_TimerSlow.ET >= T#1200MS THEN
		Sys_Variables.BlinkSlow := TRUE;  
	ELSE
		Sys_Variables.BlinkSlow := FALSE;  		
	END_IF

// ===== Always true and always false bits =====
	Sys_Variables.AlwaysOff := FALSE 	;
	Sys_Variables.AlwaysOn	:= TRUE		;
	
// ===== Manage persistent data ======
	DataManager.FbPersistentManager();

END_FUNCTION_BLOCK

// ---- Avarage/FB_RollingAverageLREAL.TcPOU
FUNCTION_BLOCK PUBLIC FB_RollingAverageLREAL
VAR_INPUT
	fInputValue	: LREAL ; // Input value [Anny_Number] 
END_VAR
VAR_IN_OUT
	bNewValue		: BOOL ; // Add value to array (set back to false)
	arLREALValues 	: ARRAY [*] OF LREAL ; // Array of LREAL values, from thich to get the average
END_VAR
VAR_OUTPUT
	fAverage	: LREAL ; // Everage of entries
END_VAR
VAR
	nWriteIndex			: DINT := 0;
	nArrayUpperBound 	: DINT;
	nArrayLowerBound 	: DINT;
	
	reNewValue	: R_TRIG ; // New value trigger
END_VAR

// determine array boundries
nArrayLowerBound := LOWER_BOUND(arLREALValues,1);
nArrayUpperBound := LOWER_BOUND(arLREALValues,1);

// Check if nwrite index is within array bounds
nWriteIndex := LIMIT(nArrayLowerBound, nWriteIndex, nArrayUpperBound);

// Add value to Array 
reNewValue(CLK := bNewValue);
IF reNewValue.Q THEN
	arLREALValues[nWriteIndex] := fInputValue;
	IF nWriteIndex = nArrayUpperBound THEN
		nWriteIndex := nArrayLowerBound;
	ELSE
		nWriteIndex := nWriteIndex +1;
	END_IF
END_IF 

// Calculate average value 
fAverage := F_AverageLREAL(arLREALValues);

METHOD PUBLIC Cmd_Reset : BOOL
VAR_INPUT
END_VAR
MEMSET(destAddr := ADR(arLREALValues), 0, n := SIZEOF(arLREALValues));
Cmd_Reset := true;
END_METHOD

END_FUNCTION_BLOCK

// ---- Avarage/F_AverageLREAL.TcPOU
FUNCTION F_AverageLREAL : LREAL
VAR_IN_OUT
	arLREALValues : ARRAY [*] OF LREAL ; // Array of LREAL values, from thich to get the average
END_VAR
VAR
	i		: DINT ;
	xSum 	: LREAL ; 
	xCount	: DINT ;
END_VAR

FOR i := LOWER_BOUND(arLREALValues,1) TO UPPER_BOUND(arLREALValues,1) DO 
	xSum 	:= arLREALValues[i] + xSum;
	xCount 	:= xCount + 1 ; 
END_FOR

IF xCount >0 THEN 
	F_AverageLREAL := xSum / xCount;
END_IF

END_FUNCTION

// ---- Avarage/FB_RollingAverageTime.TcPOU
FUNCTION_BLOCK PUBLIC FB_RollingAverageTime
VAR_INPUT
	fInputValue	: TIME ; // Input value [Anny_Number] 
END_VAR
VAR_IN_OUT
	bNewValue		: BOOL ; // Add value to array (set back to false)
	arTimeValues 	: ARRAY [*] OF TIME ; // Array of LREAL values, from thich to get the average
END_VAR
VAR_OUTPUT
	fAverage	: TIME ; // Everage of entries
END_VAR
VAR
	nWriteIndex			: DINT := 0;
	nArrayUpperBound 	: DINT;
	nArrayLowerBound 	: DINT;
	
	reNewValue	: R_TRIG ; // New value trigger
END_VAR

// determine array boundries
nArrayLowerBound := LOWER_BOUND(arTimeValues,1);
nArrayUpperBound := LOWER_BOUND(arTimeValues,1);

// Check if nwrite index is within array bounds
nWriteIndex := LIMIT(nArrayLowerBound, nWriteIndex, nArrayUpperBound);

// Add value to Array 
reNewValue(CLK := bNewValue);
IF reNewValue.Q THEN
	arTimeValues[nWriteIndex] := fInputValue;
	IF nWriteIndex = nArrayUpperBound THEN
		nWriteIndex := nArrayLowerBound;
	ELSE
		nWriteIndex := nWriteIndex +1;
	END_IF
END_IF 

// Calculate average value 
fAverage := F_AverageTime(arTimeValues);

METHOD PUBLIC Cmd_Reset : BOOL
VAR_INPUT
END_VAR
MEMSET(destAddr := ADR(arTimeValues), 0, n := SIZEOF(arTimeValues));
Cmd_Reset := true;
END_METHOD

END_FUNCTION_BLOCK

// ---- Avarage/F_AverageTime.TcPOU
FUNCTION F_AverageTime : TIME
VAR_IN_OUT
	arTimeValues : ARRAY [*] OF TIME ; // Array of LREAL values, from thich to get the average
END_VAR
VAR
	i		: DINT ;
	xSum 	: TIME ; 
	xCount	: DINT ;
END_VAR

FOR i := LOWER_BOUND(arTimeValues,1) TO UPPER_BOUND(arTimeValues,1) DO 
	xSum 	:= arTimeValues[i] + xSum;
	xCount 	:= xCount + 1 ; 
END_FOR

IF xCount >0 THEN 
	F_AverageTime := xSum / xCount;
END_IF

END_FUNCTION

// ---- BaseFunctions/FB_Base.TcPOU
FUNCTION_BLOCK PUBLIC ABSTRACT FB_Base
{attribute 'reflection'}
VAR_INPUT
	bEnable			: BOOL 		:= TRUE 	; // Module enable signal reference Default := TRUE (when using system library := GVL_Main.stModules[nModuleId].bEnabled)
	refFbParHandler	: REFERENCE TO Fb_ParLogging 	:= GVL_Parameters.fbParameterHandler	; // reference to parameter handler
	bCmdPause 		: BOOL 		:= FALSE	; // Command Pause functions		
END_VAR
VAR_IN_OUT
	refFbFault	: Fb_FaultHandler	; // reference to fault handler ( when using utilities library := GVL_Main.stModules[nModuleId].fbFaultHandler)
END_VAR
VAR_OUTPUT
	bInitOk			: BOOL 			:= FALSE 	; // function is initialized
	bBussy 			: BOOL 			:= FALSE 	; // device is busy
	bReady			: BOOL 			:= FALSE 	; // device is ready for new command 
	bErrorActive	: BOOL			:= FALSE	; // device Error active 
END_VAR
VAR
	sName			: STRING 		:= ''		; // Name of device distilled from the path 
	nLocationId		: UDINT 		:= 0		; // device id number made up of module and device number				
	
	stFault			: UDT_Fault		; // Fault data from device

	// Function path 
	{attribute 'instance-path'} 
    {attribute 'noinit'}
	sPath			: STRING	; // Path name of function (used for manual reference)
END_VAR

IF __ISVALIDREF(refFbFault) THEN 
	// check if fault is active and send to fault handler
	refFbFault.CmdAddFault(stFault);
END_IF

METHOD PUBLIC CmdReset : BOOL
VAR_INPUT
END_VAR
bErrorActive := FALSE ;

CmdReset := TRUE ;
END_METHOD

METHOD PROTECTED ExecIdentifyDevice : BOOL
VAR_INPUT
	// Message location data
	nId				: UDINT ; // Identification number of object
	nParentId		: UDINT ; // Id of higher level If aplicable (0 = no parent)
	eComponentType	: E_ComponentTypes ; // COmponent or function type for message compilation
END_VAR
// Check device ID
IF nId <> 0 AND nLocationId = 0 THEN
	nLocationId := (nParentId * 10000) + nId * 100 ;
END_IF

// set message location information
stFault.ComponentType 	:= eComponentType;
stFault.LocationName	:= F_FBNameFromPath(sPath := sPath);
stFault.LocationNumber	:= nLocationId ; 

// Get device name from function and add device to manual
IF sName = '' THEN 
	sName := F_FBNameFromPath(sPath := sPath);
END_IF

ExecIdentifyDevice := nLocationId <> 0 AND sName <> '';
END_METHOD

END_FUNCTION_BLOCK

// ---- FaultsAndMessages/Functions/Fb_FaultHandler.TcPOU
FUNCTION_BLOCK Fb_FaultHandler
VAR_INPUT
END_VAR
VAR_OUTPUT
	arActiveFaults 	: ARRAY [0..Param_Messages.nMAX_MESSAGES_SHOWN] OF UDT_Fault  ; // reference to active fault array
	nActiveFaults	: UDINT 			; // reference to active fault counter
	bActOM 			: BOOL := FALSE ;
	bActMC 			: BOOL := FALSE ;
	bActCF 			: BOOL := FALSE ;
	bActFF 			: BOOL := FALSE ;
	bActOW 			: BOOL := FALSE ;
END_VAR
VAR
	bResetting		: BOOL := FALSE ;
	// functional variables
	i 					: UDINT ;
	// fault data
	stFaultUdt 			: UDT_Fault ;
	bTimedOut 			: BOOL ; // Message has timed out
	// Message logging
	dToday				: DATE ; 
	nWriteStep			: UDINT := 0 ;
	bWriteError			: BOOL 	; // write to file error occured
	nWriteErroId		: UDINT ; // write error id
	// Write variables
	sActFileName		: STRING ;
	hFile				: UINT	:= 0;(* File handle of the source file *)
	sMessageString		: ARRAY [0..Param_Messages.nMESSAGE_COLUMNS] OF STRING (GVL_Parameters.MAX_CSV_FIELD_LENGTH); (* temporary parameter buffer to string*)
	sCSVLine			: T_MaxString := '';(* Single CSV text line (row, record), we are using string as record buffer (your are able to see created fields) *)
	sCSVField			: T_MaxString := '';(* Single CSV field value (column, record field) *)

	// Log to file functions
	fbFileOpen		: FB_FileOpen	;(* Opens file *)
	fbFileClose		: FB_FileClose	;(* Closes file *)
	fbFileGets		: FB_FileGets	;(* Reads one record (line) *)
	fbFilePuts		: FB_FilePuts	;(* Writes one record (line) *)
	fbReader		: FB_CSVMemBufferReader;(* Helper function block used to parse CSV data bytes (single record line) *)
	fbWriter		: FB_CSVMemBufferWriter;(* Helper function block used to create CSV data bytes (single record line) *)
END_VAR
VAR PERSISTENT
	dLastFileDate : DATE ;
END_VAR
VAR CONSTANT
	stEmptyMessageUdt : UDT_Fault := (	Active 			:= FALSE,
										FaultType 		:= E_FaultTypes.NA,
										MessageNumber	:= 0,
										LocationNumber	:= 0,
										Discription 	:= '',
										LocationName	:= '',
										ComponentType	:= E_ComponentTypes.NA,
										StartTime		:= DT#2020-1-1-00:00:00,
										EndTime			:= DT#2020-1-1-00:00:00,
										FullFaultId		:= '0'	)  ;
END_VAR

// Check for active faults in list
IF NOT bResetting THEN 
	ExecSetFaultBit(); 
END_IF

bResetting := FALSE ;

METHOD PRIVATE CheckEntryValid : BOOL
VAR_IN_OUT
	stFault : UDT_Fault ; // actuive fault structure input
END_VAR
VAR
	// functional variables
	i 	: UDINT ;
END_VAR
// ======= check if new entry is valid and not already active ======
CheckEntryValid S= TRUE ;
FOR i := 0 TO nActiveFaults DO
	IF arActiveFaults[i].Discription = stFault.Discription THEN 
		CheckEntryValid 			:= FALSE ; 
		arActiveFaults[i].Active 	:= TRUE ; 
	END_IF
END_FOR
END_METHOD

METHOD PUBLIC CmdAddFault : BOOL
VAR_IN_OUT
	stFault : UDT_Fault ; // active fault structure input
END_VAR
// coppy fault to internal fault udt
IF stFault.FaultType <> E_FaultTypes.NA AND stFault.Active THEN 
	// Process fault data
	IF CheckEntryValid(stFault) AND NOT bResetting THEN
		THIS^.stFaultUdt	:= stFault ;
		ExecWriteMessage();
	END_IF
	stFault 			:= stEmptyMessageUdt ;
	stFaultUdt.Active	:= FALSE ;
END_IF
END_METHOD

METHOD PUBLIC CmdReset : BOOL
VAR_INPUT
END_VAR
bResetting := TRUE ;
// Check for reset is active 
CmdReset := ExecResetFaults();
END_METHOD

METHOD PRIVATE ExecCleanUpArray : BOOL
VAR
	// functional variables
	i 					: UDINT ;
END_VAR
// Clean up array by removing blanc spaces 
FOR i := 0 TO Param_Messages.nMAX_MESSAGES_SHOWN - 1 DO 
	IF arActiveFaults[i].FaultType = 0 THEN 
		arActiveFaults[i] 	:= arActiveFaults[i+1];
		arActiveFaults[i+1] := stEmptyMessageUdt;
	END_IF
END_FOR

//Sort messages after cleaning
ExecSortMessages();
END_METHOD

METHOD PRIVATE ExecResetFaults : BOOL
VAR
	nResetPoint : UDINT := 0 ; // point of reset for active fault array (skips fault if .active bit is true)
	// functional variables
	i 					: UDINT ;
END_VAR
FOR i := 0 TO Param_Messages.nMAX_MESSAGES_SHOWN DO
	IF arActiveFaults[i].Active THEN
		CONTINUE;
	ELSE
		arActiveFaults[i] := stEmptyMessageUdt; 
	END_IF
END_FOR

ExecCleanUpArray();

bActOM 			:= FALSE;
bActMC 			:= FALSE;
bActCF 			:= FALSE;
bActFF 			:= FALSE;
bActOW 			:= FALSE;

ExecResetFaults := TRUE ;
END_METHOD

METHOD PRIVATE ExecSetFaultBit : BOOL
bActOM 	:= FALSE;
bActMC	:= FALSE;
bActCF 	:= FALSE;
bActFF 	:= FALSE;
bActOW  := FALSE;
	
FOR i := 0 TO nActiveFaults DO
	// read message type 
	CASE arActiveFaults[i].FaultType OF
		E_FaultTypes.OM : 
			IF arActiveFaults[i].Active THEN 
				bActOM 		S= TRUE ;
				
			ELSE 
				bTimedOut 	S= TRUE ;
			END_IF 
		E_FaultTypes.MC :
			IF arActiveFaults[i].Active THEN 
				bActMC 		S= TRUE ;
			ELSE 
				bTimedOut 	S= TRUE ;
			END_IF 
		E_FaultTypes.CF:
			bActCF 		S= TRUE ;
		E_FaultTypes.FF:
			bActFF 		S= TRUE ;
		E_FaultTypes.OW:
			IF arActiveFaults[i].Active THEN 
				bActOW 		S= TRUE ;
			ELSE 
				bTimedOut 	S= TRUE ;
			END_IF
			
		ELSE
			bTimedOut := FALSE ;
	END_CASE

	IF bTimedOut THEN 
		arActiveFaults[i] := stEmptyMessageUdt;				
		bTimedOut := FALSE ;
	END_IF
	// Reset active bit when timed out, if fault is still active it will be set to true again.
	arActiveFaults[i].Active R= (arActiveFaults[i].StartTime + Param_Messages.tMESSAGE_TIMEOUT) < Sys_Variables.SystemTime;
END_FOR

// clean up the fault array
ExecCleanUpArray();
END_METHOD

METHOD INTERNAL ExecSortMessages : BOOL
VAR
	k : UDINT ;
	stTempMessageStorage : UDT_Fault ; // Temporary message storage for sorting
END_VAR
FOR k := 1 TO Param_Messages.nMAX_MESSAGES_SHOWN - 1 DO 
	FOR i := 0 TO Param_Messages.nMAX_MESSAGES_SHOWN - 2 DO 
		IF arActiveFaults[i].FaultType < arActiveFaults[i+1].FaultType THEN 
			stTempMessageStorage 	:= arActiveFaults[i];
			arActiveFaults[i]		:= arActiveFaults[i+1];
			arActiveFaults[i+1]		:= stTempMessageStorage;
		END_IF
	END_FOR	 
END_FOR

ExecSortMessages := TRUE;
END_METHOD

ACTION ExecWriteMessage:
// Set message start time 
stFaultUdt.StartTime := Sys_Variables.SystemTime ;
// Fill Full Fault Id
stFaultUdt.FullFaultId := TO_STRING(stFaultUdt.FaultType);
stFaultUdt.FullFaultId := CONCAT(stFaultUdt.FullFaultId,'.');
stFaultUdt.FullFaultId := CONCAT(stFaultUdt.FullFaultId,UDINT_TO_STRING(stFaultUdt.MessageNumber));
stFaultUdt.FullFaultId := CONCAT(stFaultUdt.FullFaultId,'.');
stFaultUdt.FullFaultId := CONCAT(stFaultUdt.FullFaultId,UDINT_TO_STRING(stFaultUdt.LocationNumber));
stFaultUdt.FullFaultId := CONCAT(stFaultUdt.FullFaultId,'.');
stFaultUdt.FullFaultId := CONCAT(stFaultUdt.FullFaultId,UDINT_TO_STRING(stFaultUdt.ComponentType));
// send message to higher level 
arActiveFaults[nActiveFaults] := stFaultUdt		;
// Sort shown Massages
ExecSortMessages();
// Set pointer to next fault
IF nActiveFaults < Param_Messages.nMAX_MESSAGES_SHOWN THEN 
	nActiveFaults := nActiveFaults + 1 	;
ELSE
	nActiveFaults := 0 ;
END_IF

// Sort Messages by severity
END_ACTION

END_FUNCTION_BLOCK

// ---- PathFunctions/F_FBNameFromPath.TcPOU
FUNCTION F_FBNameFromPath : STRING // distills .fb name from function path
VAR_INPUT
	sPath	: STRING ;
END_VAR
VAR
	sTemp		: STRING ;
	nstartFbName: INT ; 
END_VAR

sTemp := sPath ;

REPEAT 
	// Look for first occurance of .fb in string
	nStartFbName := FIND( sTemp,'.fb');
	// Delete text before .fb and .fb itself
	IF nstartFbName <>0 THEN 
		sTemp := DELETE( STR := sTemp, LEN := nstartFbName + 3, 0); 
	END_IF
UNTIL
	nstartFbName = 0 
END_REPEAT

F_FBNameFromPath := sTemp ;

END_FUNCTION

// ---- BaseFunctions/FB_Base_WithEvent.TcPOU
FUNCTION_BLOCK PUBLIC ABSTRACT FB_Base_WithEvent
{attribute 'reflection'}
VAR_INPUT
	bEnable			: BOOL 		:= TRUE 	; // Module enable signal reference Default := TRUE (when using system library := GVL_Main.stModules[nModuleId].bEnabled)
	refFbParHandler	: REFERENCE TO Fb_ParLogging 	:= GVL_Parameters.fbParameterHandler	; // reference to parameter handler
	bCmdPause 		: BOOL 		:= FALSE	; // Command Pause functions		
END_VAR
VAR_OUTPUT
	bInitOk			: BOOL 			:= FALSE 	; // function is initialized
	bBussy 			: BOOL 			:= FALSE 	; // device is busy
	bReady			: BOOL 			:= FALSE 	; // device is ready for new command 
	bErrorActive	: BOOL			:= FALSE	; // device Error active 
END_VAR
VAR
	fbEvent			: FB_EventHandler 			; // Event handler for fault and message data			
	sName			: STRING 		:= ''		; // Name of device distilled from the path 
	nLocationId		: UDINT 		:= 0		; // device id number made up of module and device number				

	// Function path 
	{attribute 'instance-path'} 
    {attribute 'noinit'}
	sPath			: STRING	; // Path name of function (used for manual reference)
END_VAR

// Check for system wide errors
bErrorActive s= fbEvent.bActCF OR fbEvent.bActFF;

METHOD PUBLIC CmdReset : BOOL
VAR_INPUT
END_VAR
bErrorActive := fbEvent.CmdReset() ;

CmdReset := NOT bErrorActive ;
END_METHOD

METHOD PROTECTED ExecIdentifyDevice : BOOL
VAR_INPUT
	// Message location data
	nId				: UDINT ; // Identification number of object
	nParentId		: UDINT ; // Id of higher level If aplicable (0 = no parent)
	eComponentType	: E_ComponentTypes ; // COmponent or function type for message compilation
END_VAR
// Check device ID
IF nLocationId = 0 THEN
	nLocationId := (nParentId * 10000) + nId * 100 ;
END_IF

// Get device name from function and add device to manual
IF sName = '' THEN 
	sName := F_FBNameFromPath(sPath := sPath);
END_IF

// set message location information
fbEvent.Init ( 	sLocationName	:= sName,
				eComponentType 	:= eComponentType,
				nModuleID		:= nLocationId); 

ExecIdentifyDevice := nLocationId <> 0 AND sName <> '';
END_METHOD

END_FUNCTION_BLOCK

// ---- FaultsAndMessages/Functions/FB_EventHandler.TcPOU
FUNCTION_BLOCK PUBLIC FB_EventHandler
VAR_INPUT
	nTwincErrorId	: UDINT := 0; // OPTIONAL Error Id from twincat function block library
END_VAR
VAR_OUTPUT
	// Active events
	bActOM 			: BOOL := FALSE ;
	bActMC 			: BOOL := FALSE ;
	bActCF 			: BOOL := FALSE ;
	bActFF 			: BOOL := FALSE ;
	// Last event
	stLastEvent		: TcEventEntry 	; // Event entry discription  
END_VAR
VAR // Event Conformation data
	bConfRequired 	: BOOL := FALSE ; // Conformation of  		
	// Resetting
	bResetting		: BOOL := FALSE ;
END_VAR
VAR // location data
	// Location
	nLocationNumber	: UDINT 			:= 0; // message number array ([1]= System, [2]= Module,[3]= sub module, [4]= Component)
	sLocationName	: STRING			:= ''; // Location discription name
	eComponentType 	: E_ComponentTypes 	:= E_ComponentTypes.NA; // Part type discription
	// Module number
	nModuleID		: UDINT 			; // module reference number used for fault, enable, reset, and safety functions (default := 1, 0 = main system)
	// Source
	fbSource		: FB_TcSourceInfo;
END_VAR
VAR // Event functions 
	fbAlarm		: FB_TcAlarm ; // alarm event function
	fbMessage 	: FB_TcMessage ; // Message event
	
	hr 			: HRESULT;
	hrLastError : HRESULT;
END_VAR

METHOD PUBLIC CmdAddEvent : BOOL
VAR_INPUT
	Event			: TcEventEntry ; // Event entry discription  
END_VAR
// check if allarm has already been raised
IF fbAlarm.EqualsToEventEntryEx(stOther	:= Event) THEN
	CmdAddEvent := TRUE;
	RETURN;
END_IF

// Check Event severity
CASE Event.eSeverity OF 
	TcEventSeverity.Critical:
		bActFF 			S= TRUE ;	
		fbAlarm.CreateEx(Event,TRUE,fbSource);
		hr := fbAlarm.Raise(0);
	TcEventSeverity.Error:
		bActCF 			S= TRUE ;	
		fbAlarm.CreateEx(Event,TRUE,fbSource);
		hr := fbAlarm.Raise(0);
	TcEventSeverity.Warning:
		bActMC 			S= TRUE ;	
		fbAlarm.CreateEx(Event,FALSE,fbSource);
		hr := fbAlarm.Raise(0);
	TcEventSeverity.Info:
		bActOM 			S= TRUE ;	
		fbMessage.CreateEx(Event,fbSource);
		hr := fbMessage.Send(0);
	ELSE 
		RETURN;
END_CASE

// Add aditional error id
IF nTwincErrorId >0 THEN 
	fbAlarm.ipArguments.AddUDInt( value := nTwincErrorId);
END_IF
nTwincErrorId := 0; // Always clear error id after check

IF FAILED(hr) THEN 
	hrLastError := hr ;
ELSE
	CmdAddEvent := TRUE;
END_IF
END_METHOD

METHOD PUBLIC CmdReset : BOOL
VAR_INPUT
END_VAR
bResetting := TRUE ;

hr := fbAlarm.Clear(0,TRUE);

IF NOT FAILED(hr) THEN 
	bResetting := FALSE ; 
	bActOM 	:= FALSE ;
	bActMC	:= FALSE ;
	bActCF	:= FALSE ;
	bActFF	:= FALSE ;
END_IF

// Set feedback
CmdReset := NOT bResetting;
END_METHOD

METHOD PRIVATE ExecSetActiveEvents : BOOL
VAR_INPUT
END_VAR
END_METHOD

METHOD PUBLIC Init : BOOL
VAR_INPUT
	// Location
		sLocationName	: STRING			:= ''; // Location discription name
		eComponentType 	: E_ComponentTypes 	:= E_ComponentTypes.NA; // Part type discription
	// Module number
		nModuleID		: UDINT 			; // module reference number used for fault, enable, reset, and safety functions (default := 1, 0 = main system)
END_VAR
// Transfer location data into event location data format
fbSource.nId 	:= nModuleID;
fbSource.sName	:= TO_STRING(eComponentType);
fbSource.ExtendName(sLocationName);

fbMessage.CreateEx(TC_EVENTS.StateMessages.ModuleInitialized,fbSource);
fbMessage.Send(0);

Init := TRUE ;
END_METHOD

END_FUNCTION_BLOCK

// ---- BaseFunctions/FB_FunctionBase.TcPOU
{attribute 'reflection'}
FUNCTION_BLOCK PUBLIC ABSTRACT FB_FunctionBase EXTENDS FB_Base
VAR_INPUT
	bSafetyOk	: BOOL 		:= TRUE 				; // Module can operate safely [default true]
END_VAR
VAR_OUTPUT
	sActiveState	: STRING 		:= 'Idle'	; // active state of device 
	bManual			: BOOL 			:= FALSE 	; // device is in manual mode
	bIsSafe			: BOOL 			:= FALSE	; // Device is locked and safe
	bHeld			: BOOL 			:= FALSE 	; // Function is held
	bBlockedCommand	: BOOL 			:= FALSE 	; // a device command is blocked because of collision detect 
END_VAR
VAR
	bCmdManual 		: BOOL			:= FALSE	; // manual commands enabled control functions (thus disable automatic)
END_VAR

SUPER^(refFbFault := refFbFault);

// Communicate active state
IF NOT bSafetyOk THEN 
	sActiveState := 'Safety not ok';
ELSIF bErrorActive THEN 
	sActiveState := TO_STRING(stFault.Discription);
ELSIF NOT bInitOk THEN 
	sActiveState := 'Not initialized';
ELSIF bManual THEN 
	sActiveState := 'Manual operation';
ELSE
	sActiveState := 'Operational';
END_IF 

// check for manual command mode
bManual := bCmdManual ;

// Execute device functions
IF bInitOk THEN  
	ExecMachineSafety();
	ExecDevFunctions();
END_IF

// Set fault if commands are blocked
IF bBlockedCommand AND bHeld THEN 
	stFault.Active 			:= TRUE ;
	stFault.ComponentType 	:= E_ComponentTypes.Assembly ;
	stFault.Discription		:= CONCAT( STR1 := sName, STR2 := ' function is blocked');
	stFault.FaultType		:= E_FaultTypes.MC;
END_IF

METHOD PUBLIC CmdHold : BOOL
VAR_INPUT
END_VAR
bHeld 	:= TRUE ;
CmdHold := bHeld ;
END_METHOD

METHOD PUBLIC CmdManual : BOOL
VAR_INPUT
END_VAR
bCmdManual := true ;
END_METHOD

METHOD PUBLIC CmdSafeStop : BOOL
VAR_INPUT
END_VAR
// check if device is safe
bIsSafe 	:= NOT bEnable ;
CmdSafeStop := bIsSafe ;
END_METHOD

METHOD PROTECTED ExecDevFunctions : BOOL
VAR_INPUT
END_VAR
END_METHOD

METHOD PROTECTED ExecMachineSafety : BOOL
VAR_INPUT
END_VAR
END_METHOD

END_FUNCTION_BLOCK

// ---- BaseFunctions/FB_FunctionBase_WIthEvent.TcPOU
{attribute 'reflection'}
FUNCTION_BLOCK PUBLIC ABSTRACT FB_FunctionBase_WIthEvent EXTENDS FB_Base_WithEvent
VAR_INPUT
	bSafetyOk	: BOOL 		:= TRUE 				; // Module can operate safely [default true]
END_VAR
VAR_OUTPUT
	sActiveState	: STRING 		:= 'Idle'	; // active state of device 
	bManual			: BOOL 			:= FALSE 	; // device is in manual mode
	bIsSafe			: BOOL 			:= FALSE	; // Device is locked and safe
	bHeld			: BOOL 			:= FALSE 	; // Function is held
	bBlockedCommand	: BOOL 			:= FALSE 	; // a device command is blocked because of collision detect 
END_VAR
VAR
	bCmdManual 		: BOOL			:= FALSE	; // manual commands enabled control functions (thus disable automatic)
END_VAR

SUPER^();

// Communicate active state
IF NOT bSafetyOk THEN 
	sActiveState := 'Safety not ok';
ELSIF bErrorActive THEN 
	sActiveState := 'Error is active';
ELSIF NOT bInitOk THEN 
	sActiveState := 'Not initialized';
ELSIF bManual THEN 
	sActiveState := 'Operational';
END_IF 

// check for manual command mode
bManual := bCmdManual ;

// Execute device functions
IF bInitOk THEN  
	ExecMachineSafety();
	ExecDevFunctions();
END_IF

// Set fault if commands are blocked
IF bBlockedCommand THEN 
	fbEvent.CmdAddEvent( Event := TC_EVENTS.StateMessages.FunctionsIsBlocked);
END_IF

METHOD PUBLIC CmdHold : BOOL
VAR_INPUT
END_VAR
bHeld 	:= TRUE ;
CmdHold := bHeld ;
END_METHOD

METHOD PUBLIC CmdManual : BOOL
VAR_INPUT
END_VAR
bCmdManual := true ;
END_METHOD

METHOD PUBLIC CmdSafeStop : BOOL
VAR_INPUT
END_VAR
// check if device is safe
bIsSafe 	:= NOT bEnable ;
CmdSafeStop := bIsSafe ;
END_METHOD

METHOD PROTECTED ExecDevFunctions : BOOL
VAR_INPUT
END_VAR
END_METHOD

METHOD PROTECTED ExecMachineSafety : BOOL
VAR_INPUT
END_VAR
END_METHOD

END_FUNCTION_BLOCK

// ---- Compare/Functions/Between.TcPOU
FUNCTION Between : BOOL // Returns true if value is >= the lower and <= the upper threshold
VAR_INPUT
	Lower	: LREAL	; // lower threshold value [LREAL]
	Value	: LREAL	; // test value [LREAL]
	Upper	: LREAL	; // Upper threshold value [LREAL]
END_VAR
VAR
END_VAR

// Check if value is between lower and upper threshold
Between := (Value >= Lower) AND (Value <= Upper);

END_FUNCTION

// ---- Compare/Functions/Between360deg.TcPOU
FUNCTION Between360deg : BOOL // Returns true if value is >= the lower and <= the upper threshold, if lower > upper then upper := Upper +360 deg
VAR_INPUT
	Lower	: LREAL	; // lower threshold value [LREAL]
	Value	: LREAL	; // test value [LREAL]
	Upper	: LREAL	; // Upper threshold value [LREAL]
END_VAR
VAR
END_VAR

IF Lower > Upper THEN  
	Between360deg S= Between( Lower, Value, 360);
	Between360deg S= Between( 0, Value, Upper)	;
ELSE 
	Between360deg S= Between( Lower, Value, Upper)	;
END_IF

END_FUNCTION

// ---- Conversion/DegS_To_Rpm.TcPOU
(* convert degrees per second to rotations per minute *)
FUNCTION DegS_To_Rpm : LREAL
VAR_INPUT
	DegS : LREAL ; // Input degrees per second as long real
END_VAR

// ===== convert degrees per second to Rpm =====
	DegS_To_Rpm := (DegS/360)*60 ;

END_FUNCTION

// ---- Conversion/DegS_To_Rpm_And_MMin.TcPOU
FUNCTION DegS_To_Rpm_And_MMin : BOOL
VAR_INPUT
	DegPerSecond : LREAL ; // Input degrees per second
	StitchLength : LREAL ; // Input stitch length
END_VAR
VAR_OUTPUT
	RevPerMinute	: LREAL ; // Output revolutions per minute
	MetersPerMinute	: LREAL ; // Output meters per minute
END_VAR
VAR
END_VAR

// ===== convert degrees per second to Rpm =====
	RevPerMinute := (DegPerSecond/360)*60 ;
// ===== Convert RPM to MMin =====
	MetersPerMinute := RevPerMinute * StitchLength / 1000 ;

END_FUNCTION

// ---- Conversion/Grey_To_Bin.TcPOU
FUNCTION Grey_To_Bin : INT // convert 4 bit grey code into 8 bit binary code
VAR_INPUT
	GreyBit0 : BOOL := FALSE ;
	GreyBit1 : BOOL := FALSE ;
	GreyBit2 : BOOL := FALSE ;
	GreyBit3 : BOOL := FALSE ;
END_VAR
VAR
	TempInt : INT ; // temporary 
END_VAR

// convert grey code into binary
TempInt.3 	:= GreyBit3 ;
TempInt.2	:= GreyBit3 	XOR GreyBit2 ;
TempInt.1	:= TempInt.2	XOR GreyBit1 ;
TempInt.0	:= TempInt.1	XOR GreyBit0 ;

Grey_To_Bin := TempInt ;

END_FUNCTION

// ---- Conversion/MMin_To_Rpm_And_DegS.TcPOU
(* Convert meters per minute to degrees per second *)
FUNCTION MMin_To_Rpm_And_DegS : BOOL
VAR_INPUT
	MeterPerMinute 	: LREAL ; // Input meters per minute
	StitchLength	: LREAL ; // Input Stitch length
END_VAR
VAR_OUTPUT
	RevPerMinute	: LREAL ; // Output revolutions per minute
	DegPerSecond	: LREAL ; // Output degrees per second
END_VAR
VAR
	MmMin 	: LREAL ; // Millimeters per minute
	RevSec 	: LREAL ; // Millimeters per second
END_VAR

// ===== convert MMin to RPM =====
	RevPerMinute := (MeterPerMinute * 1000) / StitchLength ;
//===== Convert RPM to DegS =====
	DegPerSecond := (RevPerMinute/60)*360 ;

END_FUNCTION

// ---- Conversion/Rpm_To_DegS.TcPOU
(* convert rotations per minute to degrees per second *)
FUNCTION Rpm_To_DegS : LREAL 
VAR_INPUT
	Rpm : LREAL ; // input revolutions per minute
END_VAR

// ===== convert RPM to DegS ====
	Rpm_To_DegS := (Rpm/60)*360 ;

END_FUNCTION

// ---- FaultsAndMessages/Functions/FB_OperatorMessageDisplay.TcPOU
FUNCTION_BLOCK FB_OperatorMessageDisplay // function compares messages and shows latest message on screen for a set period of time
VAR_INPUT
	bEnable 	: BOOL 	:= TRUE ; // enable messages
	tDisplayTime: TIME	:= Param_Messages.tMESSAGE_TIMEOUT ; // Time before message relevance is checked (default = Param_Messages.tMESSAGE_TIMEOUT)
END_VAR
VAR_IN_OUT
	sMessage 	: STRING ; // Operator message (default = GVL_Message.sOPeratorMessage)
END_VAR
VAR_OUTPUT
	sOutMessage : STRING ; // message output to screen
END_VAR
VAR
	sOldMessage 	: STRING := ''; // old message as displayed 
	tonDisplayTimer	: TON ; // Display timer
END_VAR

// Run timers
tonDisplayTimer(PT := tDisplayTime);

// compare old message with new message 
IF sMessage = sOldMessage THEN 
	tonDisplayTimer.IN := TRUE ;
	IF tonDisplayTimer.Q = TRUE THEN 
		sMessage := '';
	END_IF
ELSE 
	tonDisplayTimer.IN 	:= FALSE 	;
	sOldMessage 		:= sMessage ; 
END_IF

// write message to display
sOutMessage := sMessage ;

END_FUNCTION_BLOCK

// ---- PathFunctions/F_GetLevelFromPath.TcPOU
FUNCTION F_GetLevelFromPath : UDINT // Get Function nesting level from path by counting '.'
VAR_INPUT
	sPath	: STRING ;
END_VAR
VAR
	sTemp		: STRING ;
	nDotPos		: INT ; 
	nLevel		: UDINT ;
END_VAR

sTemp := sPath ;

REPEAT 
	nDotPos := FIND(sTemp,'.');
	IF nDotPos <> 0 THEN 
		nLevel := nLevel +1 ;
		sTemp := DELETE(STR := sTemp,
						LEN := nDotPos + 1,
						POS	:= 0 );
	END_IF
UNTIL 
	nDotPos = 0	
END_REPEAT

F_GetLevelFromPath := nLevel;

END_FUNCTION

// ---- Positions/FunctionBlocks/FB_PositionTrigger_Old.TcPOU
FUNCTION_BLOCK PUBLIC FB_PositionTrigger_Old // trigger function, sets trigger Q signal high when trigger position is between previous cycle's and current axis position.
VAR_INPUT
	fAxisPos			: LREAL	; // Axis position on which the to trigger
	nAxisModuloRev		: DINT 	:= 0	; // axis modulo revolutions 
	fAxisVelocity		: LREAL := 0 	; 	// velocity of axis 
	bDirPositive		: BOOL 	:= TRUE ; // Axis direction is forward 
	fEncoderTurnover	: LREAL	:= 360 	; // Encoder turnover value (standard 360 deg)
	bEnablenNegative 	: BOOL 	:= FALSE; // Enables negative input values
END_VAR
VAR_OUTPUT
	Q					: BOOL 	; // trigger signal
	bInternalTrigger	: BOOL 	; // Internal trigger signal 
	bTriggerArmed 		: BOOL 	; // Trigger is armed 
	bEncoderTurnedOver	: BOOL 	; // is high when encoder goes thru it's turnover point 
	fAccuracy 			: LREAL ; // Accuracy of trigger 
END_VAR
VAR
	// function commands
	fTriggerPosition 		: LREAL ; // trigger position 
	fTriggerPosCompensated	: LREAL ; // TRigger Position after compensation
	nRotBeforeTrigger		: DINT 	:= 0 ; 	// Full axis rotations before position trigger is armed
	nRotBeforeTriggerCompensated	: DINT := 0 ; // full E_ComponentTypes.Axis rotation before trigger IsFinite armed 
	// Trigger variables 
	fReactionTime			: LREAL	:= 0 ; 	// [ms] Time before reaction to trigger (time compensation)
	// internal values	
	nTriggerRotation		: DINT	:= 0 ; 	// Number of rotations done since trigger is armed 
	fOldAxisPos				: LREAL ; 		// Old axis position for comparison
	nOldAxisRev				: DINT 	; 		// Old modulo revolutions 
	fCompensationDistance	: LREAL := 0 ; 	// [units] trigger compensation distance  
	// Edge functions 
	fbReTriggerArmed		: R_TRIG ; // rising edge trigger on trigger armed (used to rest trigger values) 
END_VAR

// Rising edge function execute
fbReTriggerArmed(CLK := bTriggerArmed); 

// ==== Skip function if trigger is not armed =====
	IF NOT bTriggerArmed THEN  
		bInternalTrigger	:= FALSE 	;
		Q 					:= FALSE	;
		RETURN ;	
	ELSIF fbReTriggerArmed.Q THEN 
		fOldAxisPos 		:= fAxisPos ;
		nOldAxisRev			:= nAxisModuloRev ;
		nTriggerRotation	:= 0 		; 
	END_IF
	
// ==== check if encoder is at turnover =====
	ExecTurnoverCheck(); 
// ==== compare positions to trigger ======
	CalcTriggerCompensation();
	ExecArmTrigger();

METHOD PRIVATE CalcTriggerCompensation : BOOL
VAR_INPUT
END_VAR
// ===== Calculate the distance travelled within the delay time =====
	fCompensationDistance	:= fReactionTime  * (fAxisVelocity / 1000);
END_METHOD

METHOD PUBLIC CmdArmTrigger : BOOL // arm trigger
VAR_INPUT
END_VAR
// Arm trigger command 
bTriggerArmed S= TRUE ;

// set feedback
CmdArmTrigger := NOT Q ;
END_METHOD

METHOD PUBLIC CmdSetTriggerPos : BOOL
VAR_INPUT
	fCmdPosition 	: LREAL ; // Trigger position 
	nCmdRotations	: DINT	:= 0 ; // Rotations before trigger is set  
	nCmdReactionTime: LREAL := 0 ; // [ms]reaction time to trigger signal 
END_VAR
// set trigger position
fTriggerPosition 	:= fCmdPosition ;
nRotBeforeTrigger	:= nCmdRotations;
fReactionTime 		:= nCmdReactionTime ;
END_METHOD

METHOD INTERNAL ExecArmTrigger : BOOL
VAR_INPUT
END_VAR
// ===== Retract compensationdistance from trigger distance =====

// check if trigger pos is not negative 
IF NOT bEnablenNegative AND fTriggerPosCompensated < 0 THEN
	fTriggerPosCompensated 			:= fEncoderTurnover + fTriggerPosition ;
	nRotBeforeTriggerCompensated	:= nRotBeforeTrigger -	1;  
ELSE
	fTriggerPosCompensated 			:= fTriggerPosition - fCompensationDistance ;
	nRotBeforeTriggerCompensated	:= nRotBeforeTrigger ;  
END_IF 

// ==== compare positions to trigger ======
	bInternalTrigger := FALSE ;

	IF bEncoderTurnedOver THEN
		IF bDirPositive THEN
			bInternalTrigger S= Between(fOldAxisPos , fTriggerPosCompensated, fEncoderTurnover) ;
			bInternalTrigger S= Between(0	, fTriggerPosCompensated, fAxisPos) ;
		ELSE 
			bInternalTrigger S= Between(0			, fTriggerPosCompensated, fOldAxisPos) ;
			bInternalTrigger S= Between(fAxisPos	, fTriggerPosCompensated, fEncoderTurnover) ;
		END_IF 
		bEncoderTurnedOver := FALSE ;
	ELSE 
		bInternalTrigger S= Between(fAxisPos	, fTriggerPosCompensated, fOldAxisPos) ;
		bInternalTrigger S= Between(fOldAxisPos	, fTriggerPosCompensated, fAxisPos) ;
		fAccuracy	:= ABS( fOldAxisPos - fAxisPos);
	END_IF

	fOldAxisPos := fAxisPos ;

// ==== Check multiturn command =======
	IF bInternalTrigger THEN 
		IF nTriggerRotation >= nRotBeforeTriggerCompensated THEN 
			Q S= bInternalTrigger OR fAxisPos > fTriggerPosCompensated;			
		ELSE 
			nTriggerRotation := nTriggerRotation + 1 ;
		END_IF 
	END_IF

// ==== Reset arm trigger command =====
	bTriggerArmed 	R= Q ;
END_METHOD

METHOD PRIVATE ExecTurnoverCheck : BOOL
VAR_INPUT
END_VAR
	bEncoderTurnedOver := nOldAxisRev <> nAxisModuloRev ;
	nOldAxisRev := nAxisModuloRev ;
END_METHOD

END_FUNCTION_BLOCK

// ---- Positions/FunctionBlocks/FB_PositionTrigger.TcPOU
FUNCTION_BLOCK PUBLIC FB_PositionTrigger // trigger function, sets trigger Q signal high when trigger position is between previous cycle's and current axis position.
VAR_INPUT
	fAxisPos			: LREAL	; // Axis position on which the to trigger
	nAxisModuloRev		: DINT 	:= 0	; // axis modulo revolutions 
	fAxisVelocity		: LREAL := 0 	; 	// velocity of axis 
	bDirPositive		: BOOL 	:= TRUE ; // Axis direction is forward 
	fEncoderTurnover	: LREAL	:= 360 	; // Encoder turnover value (standard 360 deg)
	bEnablenNegative 	: BOOL 	:= FALSE; // Enables negative input values
END_VAR
VAR_OUTPUT
	Q					: BOOL 	; // trigger signal
	bInternalTrigger	: BOOL 	; // Internal trigger signal 
	bTriggerArmed 		: BOOL 	; // Trigger is armed 
	bEncoderTurnedOver	: BOOL 	; // is high when encoder goes thru it's turnover point 
	fAccuracy 			: LREAL ; // Accuracy of trigger 
END_VAR
VAR
	// function commands
	fTriggerPosition 		: LREAL ; // trigger position 
	fTriggerPosCompensated	: LREAL ; // TRigger Position after compensation
	nRotBeforeTrigger		: DINT 	:= 0 ; 	// Full axis rotations before position trigger is armed
	nRotBeforeTriggerCompensated	: DINT := 0 ; // full E_ComponentTypes.Axis rotation before trigger IsFinite armed 
	// Trigger variables 
	fReactionTime			: LREAL	:= 0 ; 	// [ms] Time before reaction to trigger (time compensation)
	// internal values	
	nTriggerRotation		: DINT	:= 0 ; 	// Number of rotations done since trigger is armed 
	fOldAxisPos				: LREAL ; 		// Old axis position for comparison
	nOldAxisRev				: DINT 	; 		// Old modulo revolutions 
	fCompensationDistance	: LREAL := 0 ; 	// [units] trigger compensation distance  
	// Edge functions 
	fbReTriggerArmed		: R_TRIG ; // rising edge trigger on trigger armed (used to rest trigger values) 
END_VAR

// Rising edge function execute
fbReTriggerArmed(CLK := bTriggerArmed); 

// ==== Skip function if trigger is not armed =====
	IF NOT bTriggerArmed THEN  
		bInternalTrigger	:= FALSE 	;
		fOldAxisPos 		:= fAxisPos ;
		nOldAxisRev			:= nAxisModuloRev ;
		nTriggerRotation	:= 0 		; 
	END_IF
	
// ==== check if encoder is at turnover =====
	ExecTurnoverCheck(); 
// ==== compare positions to trigger ======
	CalcTriggerCompensation();
	ExecArmTrigger();

METHOD PRIVATE CalcTriggerCompensation : BOOL
VAR_INPUT
END_VAR
// ===== Calculate the distance travelled within the delay time =====
	fCompensationDistance	:= fReactionTime  * (fAxisVelocity / 1000);
END_METHOD

METHOD PUBLIC CmdArmTrigger : BOOL // arm trigger
VAR_INPUT
END_VAR
// Arm trigger command 
bTriggerArmed S= TRUE ;
Q := FALSE ;

// set feedback
CmdArmTrigger := NOT Q
 ;
END_METHOD

METHOD PUBLIC CmdSetTriggerPos : BOOL
VAR_INPUT
	fCmdPosition 	: LREAL ; // Trigger position 
	nCmdRotations	: DINT 	; // Rotations before trigger is set  
	nCmdReactionTime: LREAL ; // [ms]reaction time to trigger signal 
END_VAR
// set trigger position
fTriggerPosition 	:= fCmdPosition ;
nRotBeforeTrigger	:= nCmdRotations;
fReactionTime 		:= nCmdReactionTime ;
END_METHOD

METHOD INTERNAL ExecArmTrigger : BOOL
VAR_INPUT
END_VAR
// ===== Retract compensationdistance from trigger distance =====

// check if trigger pos is not negative 
	IF NOT bEnablenNegative AND fTriggerPosCompensated < 0 THEN
		fTriggerPosCompensated 			:= fEncoderTurnover + fTriggerPosition ;
		nRotBeforeTriggerCompensated	:= nRotBeforeTrigger -	1;  
	ELSE
		fTriggerPosCompensated 			:= fTriggerPosition - fCompensationDistance ;
		nRotBeforeTriggerCompensated	:= nRotBeforeTrigger ;  
	END_IF 

// ==== compare positions to trigger ======
	IF NOT bTriggerArmed THEN 
		bInternalTrigger := FALSE ;
	ELSIF bEncoderTurnedOver THEN
		IF bDirPositive THEN
			bInternalTrigger S= Between(fOldAxisPos , fTriggerPosCompensated, fEncoderTurnover) ;
			bInternalTrigger S= Between(0			, fTriggerPosCompensated, fAxisPos) ;
		ELSE 
			bInternalTrigger S= Between(0			, fTriggerPosCompensated, fOldAxisPos) ;
			bInternalTrigger S= Between(fAxisPos	, fTriggerPosCompensated, fEncoderTurnover) ;
		END_IF 
		bEncoderTurnedOver := FALSE ;
	ELSE 
		bInternalTrigger S= Between(fAxisPos	, fTriggerPosCompensated, fOldAxisPos) ;
		bInternalTrigger S= Between(fOldAxisPos	, fTriggerPosCompensated, fAxisPos) ;
		fAccuracy	:= ABS( fOldAxisPos - fAxisPos);
	END_IF

	fOldAxisPos := fAxisPos ;

// ==== Check multiturn command =======
	IF bInternalTrigger THEN 
		IF nTriggerRotation >= nRotBeforeTriggerCompensated THEN 
			Q := bInternalTrigger OR fAxisPos > fTriggerPosCompensated;
			bTriggerArmed := FALSE ;			
		ELSE 
			nTriggerRotation := nTriggerRotation + 1 ;
		END_IF 
		bInternalTrigger := FALSE ;
	ELSE 
		Q:= FALSE ;
	END_IF
END_METHOD

METHOD PRIVATE ExecTurnoverCheck : BOOL
VAR_INPUT
END_VAR
	bEncoderTurnedOver 	:= nOldAxisRev <> nAxisModuloRev ;
	nOldAxisRev 		:= nAxisModuloRev ;
END_METHOD

END_FUNCTION_BLOCK

// ---- Positions/Functions/F_AccDecDistanceFromTime.TcPOU
FUNCTION F_AccDecDistanceFromTime : LREAL
VAR_INPUT
	nAccelDecel	: LREAL ; // acceleration or deceleration [units/s^2]
	nTimeMs		: LREAL	; // Time for acceleratio/ deceleration to take place [ms]
END_VAR
VAR
	nTimeSec	: LREAL;
	nVelocity	: LREAL;
END_VAR

nTimeSec := nTimeMs/1000;

nVelocity := nAccelDecel * nTimeSec;

F_AccDecDistanceFromTime := nVelocity * nTimeSec / 2 ;

END_FUNCTION

// ---- Positions/Functions/F_AccDecDistanceFromVelo.TcPOU
FUNCTION F_AccDecDistanceFromVelo : LREAL
VAR_INPUT
	nVelocity	: LREAL ; // velocity [m/s]
	nAccDecc	: LREAL ; // acceleration or deceleration value [m/s^2]
END_VAR
VAR
	nTime : LREAL ;
END_VAR

nTime := nVelocity	/	nAccDecc ;

F_AccDecDistanceFromVelo := nVelocity * (nTime/2);

END_FUNCTION

// ---- Positions/Functions/F_PosCheck.TcPOU
(* Returns a true when position is within tollerance *)
FUNCTION F_PosCheck : bool
VAR_INPUT
	TargetPos		: LREAL ; // target position to check [deg]
	ActPos			: LREAL	; // Actual position [deg]
	Lowtol			: LREAL	; // Low tolerance (is reduced from target pos)
	HighTol			: LREAL	; // High tollerance (is added to target position)
	EncTurnover		: DINT 	; // Encoder turnover value
END_VAR
VAR
	Lowval	: LREAL ;
	HighVal	: LREAL ;
	LowTurn	: BOOL ;
	HighTurn: BOOL ;
	HighOk	: BOOL ;
	LowOK	: BOOL ;
END_VAR

// Check lower and uper do not exceed turnover
	IF TargetPos - Lowtol < 0 THEN 
		Lowval 	:= EncTurnover + TargetPos - Lowtol ;
		LowTurn	:= TRUE ;
	ELSE 
		LowTurn := FALSE ;
	END_IF

	IF TargetPos + HighTol > 360 THEN 
		HighVal	:= EncTurnover - TargetPos + Lowtol ;
		HighTurn:= TRUE ;
	ELSE 
		HighTurn := FALSE ;
	END_IF

	
// Check lower limit
	IF LowTurn AND ActPos > Lowval THEN
		LowOK := TRUE ; 
	ELSIF HighTurn AND ActPos < HighVal THEN 
		LowOK := TRUE ;
	ELSIF ActPos > TargetPos - Lowtol THEN
		LowOK := TRUE ;
	ELSE 
		LowOK := FALSE ;
	END_IF
	
// Check high limit
	IF HighTurn AND ActPos < HighVal THEN
		HighOk := TRUE ;
	ELSIF LowTurn AND ActPos > Lowval THEN 
		HighOk := TRUE ; 
	ELSIF ActPos < TargetPos + HighTol THEN
		HighOk := TRUE ;
	ELSE
		HighOk := FALSE ;
	END_IF
	
// Set output
	IF LowOK AND HighOk THEN
		F_PosCheck := TRUE ;
	ELSE 
		F_PosCheck := FALSE ;
	END_IF

END_FUNCTION

// ---- Positions/Functions/F_TopVelocityFromTime.TcPOU
FUNCTION F_TopVelocityFromTime : LREAL
VAR_INPUT
	nAccel	: LREAL ; // acceleration or deceleration [units/s^2]
	nTimeMs		: LREAL	; // Time for acceleratio/ deceleration to take place [ms]
END_VAR
VAR
	nTimeSec	: LREAL;
END_VAR

nTimeSec := nTimeMs/1000;

F_TopVelocityFromTime := nAccel * nTimeSec;

END_FUNCTION

// ---- Positions/Functions/F_TriggerPosOffset.TcPOU
(* function to calculate trigger points for time based moves *)
FUNCTION F_TriggerPosOffset : LREAL
VAR_INPUT
	Velocity		: LREAL	; // [Units/sec] command velocity 
	nMoveTimeMs		: LREAL	; // [ms] Time it takes for move to complete
END_VAR
VAR
END_VAR

// ===== Convert time to usable calculation value =====
	F_TriggerPosOffset := nMovetimeMs * ABS(Velocity / 1000);

END_FUNCTION

// ---- StepFunctions/FB_Step.TcPOU
FUNCTION_BLOCK PUBLIC FB_Step EXTENDS FB_Base_WithEvent
VAR_INPUT
END_VAR
VAR_OUTPUT
	nActStep	: UDINT := 0 ; // Active step
	bIdle		: BOOL	:= TRUE  ; // Stepper is idle (Step 0)
	bPaused		: BOOL 	:= FALSE ; // Stepper is paused
	bHold		: BOOL 	:= FALSE ; // Stepper is blocked for changes
	bSkipPause	: BOOL	:= FALSE ; // Pause function is skipped in this step 
	bResetting	: BOOL  := False ; // Reset is active
END_VAR
VAR
	nPreviousStep 	: UDINT ; // Previous active step
	nNextStep		: UDINT ; // Next step to activate
	nResetStep		: UDINT ; // step to which the stepper will go after reset
END_VAR

SetActiveStep();

METHOD PUBLIC CmdHold : BOOL
VAR_INPUT
END_VAR
bHold := TRUE ;

CmdHold := bHold;
END_METHOD

METHOD PUBLIC CmdNext : BOOL
VAR_INPUT
END_VAR
IF NOT bHold THEN 
	nNextStep := nActStep +	1 ;	
END_IF

CmdNext := TRUE ;
END_METHOD

METHOD PUBLIC CmdPrevious : BOOL
VAR_INPUT
END_VAR
IF NOT bHold THEN 
	nNextStep := nPreviousStep ;	
END_IF

CmdPrevious := TRUE ;
END_METHOD

METHOD PUBLIC CmdReset : BOOL
VAR_INPUT
END_VAR
bErrorActive := FALSE ;

IF nActStep <> nResetStep THEN 
	IF NOT bResetting THEN
		bResetting := TRUE ;
	ELSE
		nPreviousStep 	:= nActStep ;
		nNextStep		:= nResetStep ;
		nActStep 		:= nResetStep ;
		bResetting 		:= FALSE;
	END_IF
ELSE
	CmdReset := TRUE ; 
END_IF
END_METHOD

METHOD PUBLIC CmdToStep : BOOL
VAR_INPUT
	nStep	: UDINT ;
END_VAR
IF NOT bHold THEN 
	nNextStep := nStep ;
END_IF

CmdToStep := nNextStep = nStep ;
END_METHOD

METHOD PUBLIC Init : BOOL
VAR_INPUT
	// Location data for messages  
	nId			: UDINT ; // Identification number of object
	nParentId	: UDINT ; // Id of higher level If aplicable (0 = no parent)
	nResetStep	: UDINT ; // step to which the stepper wil go at reset
END_VAR
// ====== Calculate device id =====
	ExecIdentifyDevice(nId,nParentId,E_ComponentTypes.StepProgram);
	
// ===== set reset step ======
	nActStep 			:= nResetStep ;
	THIS^.nResetStep	:= nResetStep ;
END_METHOD

METHOD PRIVATE SetActiveStep : BOOL
VAR_INPUT
END_VAR
IF bResetting THEN 
	nPreviousStep 	:= nActStep ;
	nNextStep		:= nResetStep ;
	nActStep 		:= nResetStep ;
	bResetting 		:= FALSE; 
ELSIF bHold THEN 
	bHold 			:= FALSE ;
	RETURN; 
ELSIF bErrorActive THEN 
	fbEvent.CmdAddEvent(Event := TC_EVENTS.ProgramEvents.StepNotDefined);
ELSIF NOT bCmdPause OR bSkipPause THEN 
	IF nActStep <> nNextStep THEN 
		nPreviousStep 	:=	nActStep;	
		nActStep		:= 	nNextStep;
	END_IF
END_IF

bPaused 	:= bCmdPause ;	
bSkipPause 	:= FALSE ; 
bIdle 		:= nActStep = 0 ;
END_METHOD

METHOD Public SkipPause : BOOL
VAR_INPUT
END_VAR
bSkipPause := TRUE ;

SkipPause := true ;
END_METHOD

METHOD PUBLIC StepError : BOOL
VAR_INPUT
END_VAR
bErrorActive := TRUE ;
END_METHOD

END_FUNCTION_BLOCK
